    (* Table initialization: fTable_Al *)
    fTable_Al[0, 0] := 10.0000; fTable_Al[0, 1] := -9999; fTable_Al[0, 2] := 3.11990;
    fTable_Al[1, 0] := 10.1617; fTable_Al[1, 1] := -9999; fTable_Al[1, 2] := 3.05822;
    fTable_Al[2, 0] := 10.3261; fTable_Al[2, 1] := -9999; fTable_Al[2, 2] := 2.99776;
    fTable_Al[3, 0] := 10.4931; fTable_Al[3, 1] := -9999; fTable_Al[3, 2] := 2.93850;
    fTable_Al[4, 0] := 10.6628; fTable_Al[4, 1] := -9999; fTable_Al[4, 2] := 2.88041;
    fTable_Al[5, 0] := 10.8353; fTable_Al[5, 1] := -9999; fTable_Al[5, 2] := 2.82347;
    fTable_Al[6, 0] := 11.0106; fTable_Al[6, 1] := -9999; fTable_Al[6, 2] := 2.76766;
    fTable_Al[7, 0] := 11.1886; fTable_Al[7, 1] := -9999; fTable_Al[7, 2] := 2.72200;
    fTable_Al[8, 0] := 11.3696; fTable_Al[8, 1] := -9999; fTable_Al[8, 2] := 2.69148;
    fTable_Al[9, 0] := 11.5535; fTable_Al[9, 1] := -9999; fTable_Al[9, 2] := 2.66129;
    fTable_Al[10, 0] := 11.7404; fTable_Al[10, 1] := -9999; fTable_Al[10, 2] := 2.63145;
    fTable_Al[11, 0] := 11.9303; fTable_Al[11, 1] := -9999; fTable_Al[11, 2] := 2.60195;
    fTable_Al[12, 0] := 12.1232; fTable_Al[12, 1] := -9999; fTable_Al[12, 2] := 2.57277;
    fTable_Al[13, 0] := 12.3193; fTable_Al[13, 1] := -9999; fTable_Al[13, 2] := 2.54392;
    fTable_Al[14, 0] := 12.5186; fTable_Al[14, 1] := -9999; fTable_Al[14, 2] := 2.51539;
    fTable_Al[15, 0] := 12.7210; fTable_Al[15, 1] := -9999; fTable_Al[15, 2] := 2.46668;
    fTable_Al[16, 0] := 12.9268; fTable_Al[16, 1] := -9999; fTable_Al[16, 2] := 2.41373;
    fTable_Al[17, 0] := 13.1359; fTable_Al[17, 1] := -9999; fTable_Al[17, 2] := 2.36192;
    fTable_Al[18, 0] := 13.3483; fTable_Al[18, 1] := -9999; fTable_Al[18, 2] := 2.30898;
    fTable_Al[19, 0] := 13.5642; fTable_Al[19, 1] := -9999; fTable_Al[19, 2] := 2.23405;
    fTable_Al[20, 0] := 13.7836; fTable_Al[20, 1] := -9999; fTable_Al[20, 2] := 2.15356;
    fTable_Al[21, 0] := 14.0066; fTable_Al[21, 1] := -9999; fTable_Al[21, 2] := 2.06069;
    fTable_Al[22, 0] := 14.2331; fTable_Al[22, 1] := -9999; fTable_Al[22, 2] := 1.96756;
    fTable_Al[23, 0] := 14.4633; fTable_Al[23, 1] := -9999; fTable_Al[23, 2] := 1.81305;
    fTable_Al[24, 0] := 14.6973; fTable_Al[24, 1] := -9999; fTable_Al[24, 2] := 1.35947;
    fTable_Al[25, 0] := 14.9350; fTable_Al[25, 1] := -9999; fTable_Al[25, 2] := 0.902011;
    fTable_Al[26, 0] := 15.1765; fTable_Al[26, 1] := -9999; fTable_Al[26, 2] := 0.609172;
    fTable_Al[27, 0] := 15.4220; fTable_Al[27, 1] := -9999; fTable_Al[27, 2] := 0.439681;
    fTable_Al[28, 0] := 15.6714; fTable_Al[28, 1] := -9999; fTable_Al[28, 2] := 0.372037;
    fTable_Al[29, 0] := 15.9249; fTable_Al[29, 1] := -9999; fTable_Al[29, 2] := 0.326005;
    fTable_Al[30, 0] := 16.1825; fTable_Al[30, 1] := -9999; fTable_Al[30, 2] := 0.285669;
    fTable_Al[31, 0] := 16.4442; fTable_Al[31, 1] := -9999; fTable_Al[31, 2] := 0.247205;
    fTable_Al[32, 0] := 16.7102; fTable_Al[32, 1] := -9999; fTable_Al[32, 2] := 0.213520;
    fTable_Al[33, 0] := 16.9805; fTable_Al[33, 1] := -9999; fTable_Al[33, 2] := 0.196522;
    fTable_Al[34, 0] := 17.2551; fTable_Al[34, 1] := -9999; fTable_Al[34, 2] := 0.181095;
    fTable_Al[35, 0] := 17.5342; fTable_Al[35, 1] := -9999; fTable_Al[35, 2] := 0.168385;
    fTable_Al[36, 0] := 17.8178; fTable_Al[36, 1] := -9999; fTable_Al[36, 2] := 0.160808;
    fTable_Al[37, 0] := 18.1060; fTable_Al[37, 1] := -9999; fTable_Al[37, 2] := 0.153573;
    fTable_Al[38, 0] := 18.3989; fTable_Al[38, 1] := -9999; fTable_Al[38, 2] := 0.146663;
    fTable_Al[39, 0] := 18.6964; fTable_Al[39, 1] := -9999; fTable_Al[39, 2] := 0.140063;
    fTable_Al[40, 0] := 18.9988; fTable_Al[40, 1] := -9999; fTable_Al[40, 2] := 0.133164;
    fTable_Al[41, 0] := 19.3061; fTable_Al[41, 1] := -9999; fTable_Al[41, 2] := 0.126575;
    fTable_Al[42, 0] := 19.6184; fTable_Al[42, 1] := -9999; fTable_Al[42, 2] := 0.120312;
    fTable_Al[43, 0] := 19.9357; fTable_Al[43, 1] := -9999; fTable_Al[43, 2] := 0.114360;
    fTable_Al[44, 0] := 20.2582; fTable_Al[44, 1] := -9999; fTable_Al[44, 2] := 0.109752;
    fTable_Al[45, 0] := 20.5858; fTable_Al[45, 1] := -9999; fTable_Al[45, 2] := 0.111010;
    fTable_Al[46, 0] := 20.9188; fTable_Al[46, 1] := -9999; fTable_Al[46, 2] := 0.112282;
    fTable_Al[47, 0] := 21.2571; fTable_Al[47, 1] := -9999; fTable_Al[47, 2] := 0.113569;
    fTable_Al[48, 0] := 21.6009; fTable_Al[48, 1] := -9999; fTable_Al[48, 2] := 0.114870;
    fTable_Al[49, 0] := 21.9503; fTable_Al[49, 1] := -9999; fTable_Al[49, 2] := 0.116186;
    fTable_Al[50, 0] := 22.3053; fTable_Al[50, 1] := -9999; fTable_Al[50, 2] := 0.117518;
    fTable_Al[51, 0] := 22.6661; fTable_Al[51, 1] := -9999; fTable_Al[51, 2] := 0.118864;
    fTable_Al[52, 0] := 23.0327; fTable_Al[52, 1] := -9999; fTable_Al[52, 2] := 0.120227;
    fTable_Al[53, 0] := 23.4053; fTable_Al[53, 1] := -9999; fTable_Al[53, 2] := 0.122751;
    fTable_Al[54, 0] := 23.7838; fTable_Al[54, 1] := -9999; fTable_Al[54, 2] := 0.126315;
    fTable_Al[55, 0] := 24.1685; fTable_Al[55, 1] := -9999; fTable_Al[55, 2] := 0.129984;
    fTable_Al[56, 0] := 24.5594; fTable_Al[56, 1] := -9999; fTable_Al[56, 2] := 0.133759;
    fTable_Al[57, 0] := 24.9566; fTable_Al[57, 1] := -9999; fTable_Al[57, 2] := 0.137643;
    fTable_Al[58, 0] := 25.3603; fTable_Al[58, 1] := -9999; fTable_Al[58, 2] := 0.141640;
    fTable_Al[59, 0] := 25.7705; fTable_Al[59, 1] := -9999; fTable_Al[59, 2] := 0.145495;
    fTable_Al[60, 0] := 26.1873; fTable_Al[60, 1] := -9999; fTable_Al[60, 2] := 0.148244;
    fTable_Al[61, 0] := 26.6109; fTable_Al[61, 1] := -9999; fTable_Al[61, 2] := 0.151045;
    fTable_Al[62, 0] := 27.0413; fTable_Al[62, 1] := -9999; fTable_Al[62, 2] := 0.153898;
    fTable_Al[63, 0] := 27.4786; fTable_Al[63, 1] := -9999; fTable_Al[63, 2] := 0.156806;
    fTable_Al[64, 0] := 27.9231; fTable_Al[64, 1] := -9999; fTable_Al[64, 2] := 0.159768;
    fTable_Al[65, 0] := 28.3747; fTable_Al[65, 1] := -9999; fTable_Al[65, 2] := 0.162787;
    fTable_Al[66, 0] := 28.8337; fTable_Al[66, 1] := -9999; fTable_Al[66, 2] := 0.165863;
    fTable_Al[67, 0] := 29.3000; fTable_Al[67, 1] := 2.34285; fTable_Al[67, 2] := 0.168996;
    fTable_Al[68, 0] := 29.7739; fTable_Al[68, 1] := 2.32717; fTable_Al[68, 2] := 0.172189;
    fTable_Al[69, 0] := 30.2555; fTable_Al[69, 1] := 2.31139; fTable_Al[69, 2] := 0.175442;
    fTable_Al[70, 0] := 30.7449; fTable_Al[70, 1] := 2.29552; fTable_Al[70, 2] := 0.178757;
    fTable_Al[71, 0] := 31.2421; fTable_Al[71, 1] := 2.27956; fTable_Al[71, 2] := 0.182134;
    fTable_Al[72, 0] := 31.7475; fTable_Al[72, 1] := 2.26350; fTable_Al[72, 2] := 0.185575;
    fTable_Al[73, 0] := 32.2609; fTable_Al[73, 1] := 2.24754; fTable_Al[73, 2] := 0.189081;
    fTable_Al[74, 0] := 32.7827; fTable_Al[74, 1] := 2.23175; fTable_Al[74, 2] := 0.192378;
    fTable_Al[75, 0] := 33.3130; fTable_Al[75, 1] := 2.21555; fTable_Al[75, 2] := 0.194561;
    fTable_Al[76, 0] := 33.8518; fTable_Al[76, 1] := 2.19843; fTable_Al[76, 2] := 0.196767;
    fTable_Al[77, 0] := 34.3993; fTable_Al[77, 1] := 2.18068; fTable_Al[77, 2] := 0.198999;
    fTable_Al[78, 0] := 34.9557; fTable_Al[78, 1] := 2.16235; fTable_Al[78, 2] := 0.201256;
    fTable_Al[79, 0] := 35.5211; fTable_Al[79, 1] := 2.14342; fTable_Al[79, 2] := 0.203539;
    fTable_Al[80, 0] := 36.0956; fTable_Al[80, 1] := 2.12388; fTable_Al[80, 2] := 0.205847;
    fTable_Al[81, 0] := 36.6794; fTable_Al[81, 1] := 2.10371; fTable_Al[81, 2] := 0.208182;
    fTable_Al[82, 0] := 37.2727; fTable_Al[82, 1] := 2.08287; fTable_Al[82, 2] := 0.210544;
    fTable_Al[83, 0] := 37.8755; fTable_Al[83, 1] := 2.06135; fTable_Al[83, 2] := 0.212932;
    fTable_Al[84, 0] := 38.4882; fTable_Al[84, 1] := 2.03911; fTable_Al[84, 2] := 0.215347;
    fTable_Al[85, 0] := 39.1107; fTable_Al[85, 1] := 2.01612; fTable_Al[85, 2] := 0.217789;
    fTable_Al[86, 0] := 39.7432; fTable_Al[86, 1] := 1.99237; fTable_Al[86, 2] := 0.220259;
    fTable_Al[87, 0] := 40.3861; fTable_Al[87, 1] := 1.96797; fTable_Al[87, 2] := 0.222758;
    fTable_Al[88, 0] := 41.0393; fTable_Al[88, 1] := 1.94295; fTable_Al[88, 2] := 0.225068;
    fTable_Al[89, 0] := 41.7031; fTable_Al[89, 1] := 1.91682; fTable_Al[89, 2] := 0.226470;
    fTable_Al[90, 0] := 42.3776; fTable_Al[90, 1] := 1.88912; fTable_Al[90, 2] := 0.227880;
    fTable_Al[91, 0] := 43.0630; fTable_Al[91, 1] := 1.86007; fTable_Al[91, 2] := 0.229299;
    fTable_Al[92, 0] := 43.7595; fTable_Al[92, 1] := 1.82966; fTable_Al[92, 2] := 0.230727;
    fTable_Al[93, 0] := 44.4673; fTable_Al[93, 1] := 1.79787; fTable_Al[93, 2] := 0.232164;
    fTable_Al[94, 0] := 45.1865; fTable_Al[94, 1] := 1.76466; fTable_Al[94, 2] := 0.233610;
    fTable_Al[95, 0] := 45.9174; fTable_Al[95, 1] := 1.73005; fTable_Al[95, 2] := 0.235064;
    fTable_Al[96, 0] := 46.6600; fTable_Al[96, 1] := 1.69399; fTable_Al[96, 2] := 0.236528;
    fTable_Al[97, 0] := 47.4147; fTable_Al[97, 1] := 1.65814; fTable_Al[97, 2] := 0.238001;
    fTable_Al[98, 0] := 48.1816; fTable_Al[98, 1] := 1.62074; fTable_Al[98, 2] := 0.235842;
    fTable_Al[99, 0] := 48.9609; fTable_Al[99, 1] := 1.57843; fTable_Al[99, 2] := 0.232104;
    fTable_Al[100, 0] := 49.7528; fTable_Al[100, 1] := 1.53229; fTable_Al[100, 2] := 0.228425;
    fTable_Al[101, 0] := 50.5576; fTable_Al[101, 1] := 1.48252; fTable_Al[101, 2] := 0.224805;
    fTable_Al[102, 0] := 51.3753; fTable_Al[102, 1] := 1.42904; fTable_Al[102, 2] := 0.221242;
    fTable_Al[103, 0] := 52.2062; fTable_Al[103, 1] := 1.37159; fTable_Al[103, 2] := 0.217735;
    fTable_Al[104, 0] := 53.0506; fTable_Al[104, 1] := 1.30972; fTable_Al[104, 2] := 0.214284;
    fTable_Al[105, 0] := 53.9087; fTable_Al[105, 1] := 1.24315; fTable_Al[105, 2] := 0.211759;
    fTable_Al[106, 0] := 54.7806; fTable_Al[106, 1] := 1.17229; fTable_Al[106, 2] := 0.209829;
    fTable_Al[107, 0] := 55.6667; fTable_Al[107, 1] := 1.09675; fTable_Al[107, 2] := 0.207917;
    fTable_Al[108, 0] := 56.5670; fTable_Al[108, 1] := 1.01559; fTable_Al[108, 2] := 0.206022;
    fTable_Al[109, 0] := 57.4820; fTable_Al[109, 1] := 0.928103; fTable_Al[109, 2] := 0.204145;
    fTable_Al[110, 0] := 58.4117; fTable_Al[110, 1] := 0.833427; fTable_Al[110, 2] := 0.202284;
    fTable_Al[111, 0] := 59.3564; fTable_Al[111, 1] := 0.729805; fTable_Al[111, 2] := 0.200441;
    fTable_Al[112, 0] := 60.3165; fTable_Al[112, 1] := 0.616720; fTable_Al[112, 2] := 0.200207;
    fTable_Al[113, 0] := 61.2921; fTable_Al[113, 1] := 0.494009; fTable_Al[113, 2] := 0.200602;
    fTable_Al[114, 0] := 62.2834; fTable_Al[114, 1] := 0.359171; fTable_Al[114, 2] := 0.200998;
    fTable_Al[115, 0] := 63.2908; fTable_Al[115, 1] := 0.206766; fTable_Al[115, 2] := 0.201394;
    fTable_Al[116, 0] := 64.3145; fTable_Al[116, 1] := 0.0367838; fTable_Al[116, 2] := 0.208215;
    fTable_Al[117, 0] := 65.3547; fTable_Al[117, 1] := -0.150100; fTable_Al[117, 2] := 0.215821;
    fTable_Al[118, 0] := 66.4118; fTable_Al[118, 1] := -0.363400; fTable_Al[118, 2] := 0.223705;
    fTable_Al[119, 0] := 67.4859; fTable_Al[119, 1] := -0.612251; fTable_Al[119, 2] := 0.231878;
    fTable_Al[120, 0] := 68.5775; fTable_Al[120, 1] := -0.913185; fTable_Al[120, 2] := 0.239512;
    fTable_Al[121, 0] := 69.6867; fTable_Al[121, 1] := -1.29772; fTable_Al[121, 2] := 0.247287;
    fTable_Al[122, 0] := 70.8138; fTable_Al[122, 1] := -1.83916; fTable_Al[122, 2] := 0.255315;
    fTable_Al[123, 0] := 71.9591; fTable_Al[123, 1] := -2.82640; fTable_Al[123, 2] := 0.263603;
    fTable_Al[124, 0] := 72.6000; fTable_Al[124, 1] := -4.71870; fTable_Al[124, 2] := 0.268298;
    fTable_Al[125, 0] := 72.8000; fTable_Al[125, 1] := -4.77865; fTable_Al[125, 2] := 3.05391;
    fTable_Al[126, 0] := 73.1230; fTable_Al[126, 1] := -3.57738; fTable_Al[126, 2] := 3.10106;
    fTable_Al[127, 0] := 74.3057; fTable_Al[127, 1] := -2.58986; fTable_Al[127, 2] := 3.27808;
    fTable_Al[128, 0] := 75.5076; fTable_Al[128, 1] := -2.24498; fTable_Al[128, 2] := 3.46521;
    fTable_Al[129, 0] := 76.7289; fTable_Al[129, 1] := -2.04974; fTable_Al[129, 2] := 3.66301;
    fTable_Al[130, 0] := 77.9699; fTable_Al[130, 1] := -1.91658; fTable_Al[130, 2] := 3.87212;
    fTable_Al[131, 0] := 79.2310; fTable_Al[131, 1] := -1.81173; fTable_Al[131, 2] := 4.09316;
    fTable_Al[132, 0] := 80.5125; fTable_Al[132, 1] := -1.71207; fTable_Al[132, 2] := 4.32681;
    fTable_Al[133, 0] := 81.8147; fTable_Al[133, 1] := -1.61278; fTable_Al[133, 2] := 4.55877;
    fTable_Al[134, 0] := 83.1380; fTable_Al[134, 1] := -1.51695; fTable_Al[134, 2] := 4.80227;
    fTable_Al[135, 0] := 84.4827; fTable_Al[135, 1] := -1.40821; fTable_Al[135, 2] := 5.05877;
    fTable_Al[136, 0] := 85.8491; fTable_Al[136, 1] := -1.24639; fTable_Al[136, 2] := 5.32897;
    fTable_Al[137, 0] := 87.2377; fTable_Al[137, 1] := -1.04412; fTable_Al[137, 2] := 5.54566;
    fTable_Al[138, 0] := 88.6487; fTable_Al[138, 1] := -0.869623; fTable_Al[138, 2] := 5.69070;
    fTable_Al[139, 0] := 90.0825; fTable_Al[139, 1] := -0.729715; fTable_Al[139, 2] := 5.83953;
    fTable_Al[140, 0] := 91.5395; fTable_Al[140, 1] := -0.602517; fTable_Al[140, 2] := 5.99225;
    fTable_Al[141, 0] := 93.0201; fTable_Al[141, 1] := -0.481649; fTable_Al[141, 2] := 6.14897;
    fTable_Al[142, 0] := 94.5246; fTable_Al[142, 1] := -0.363849; fTable_Al[142, 2] := 6.30978;
    fTable_Al[143, 0] := 96.0535; fTable_Al[143, 1] := -0.246485; fTable_Al[143, 2] := 6.47480;
    fTable_Al[144, 0] := 97.6071; fTable_Al[144, 1] := -0.127798; fTable_Al[144, 2] := 6.64413;
    fTable_Al[145, 0] := 99.1858; fTable_Al[145, 1] := -0.00572152; fTable_Al[145, 2] := 6.81790;
    fTable_Al[146, 0] := 100.790; fTable_Al[146, 1] := 0.121587; fTable_Al[146, 2] := 6.99620;
    fTable_Al[147, 0] := 102.420; fTable_Al[147, 1] := 0.257648; fTable_Al[147, 2] := 7.17918;
    fTable_Al[148, 0] := 104.077; fTable_Al[148, 1] := 0.408417; fTable_Al[148, 2] := 7.36022;
    fTable_Al[149, 0] := 105.760; fTable_Al[149, 1] := 0.563135; fTable_Al[149, 2] := 7.52866;
    fTable_Al[150, 0] := 107.471; fTable_Al[150, 1] := 0.713525; fTable_Al[150, 2] := 7.70096;
    fTable_Al[151, 0] := 109.209; fTable_Al[151, 1] := 0.869599; fTable_Al[151, 2] := 7.87720;
    fTable_Al[152, 0] := 110.975; fTable_Al[152, 1] := 1.03257; fTable_Al[152, 2] := 8.05748;
    fTable_Al[153, 0] := 112.770; fTable_Al[153, 1] := 1.20465; fTable_Al[153, 2] := 8.24188;
    fTable_Al[154, 0] := 114.594; fTable_Al[154, 1] := 1.38785; fTable_Al[154, 2] := 8.43050;
    fTable_Al[155, 0] := 116.448; fTable_Al[155, 1] := 1.58511; fTable_Al[155, 2] := 8.62344;
    fTable_Al[156, 0] := 118.331; fTable_Al[156, 1] := 1.79993; fTable_Al[156, 2] := 8.82080;
    fTable_Al[157, 0] := 120.245; fTable_Al[157, 1] := 2.03832; fTable_Al[157, 2] := 9.02267;
    fTable_Al[158, 0] := 122.190; fTable_Al[158, 1] := 2.31105; fTable_Al[158, 2] := 9.22916;
    fTable_Al[159, 0] := 124.166; fTable_Al[159, 1] := 2.65726; fTable_Al[159, 2] := 9.44037;
    fTable_Al[160, 0] := 126.175; fTable_Al[160, 1] := 3.05450; fTable_Al[160, 2] := 9.49754;
    fTable_Al[161, 0] := 128.215; fTable_Al[161, 1] := 3.37636; fTable_Al[161, 2] := 9.51114;
    fTable_Al[162, 0] := 130.289; fTable_Al[162, 1] := 3.65455; fTable_Al[162, 2] := 9.52475;
    fTable_Al[163, 0] := 132.397; fTable_Al[163, 1] := 3.91635; fTable_Al[163, 2] := 9.53840;
    fTable_Al[164, 0] := 134.538; fTable_Al[164, 1] := 4.16654; fTable_Al[164, 2] := 9.55206;
    fTable_Al[165, 0] := 136.714; fTable_Al[165, 1] := 4.40886; fTable_Al[165, 2] := 9.56573;
    fTable_Al[166, 0] := 138.925; fTable_Al[166, 1] := 4.64594; fTable_Al[166, 2] := 9.57943;
    fTable_Al[167, 0] := 141.172; fTable_Al[167, 1] := 4.87987; fTable_Al[167, 2] := 9.59315;
    fTable_Al[168, 0] := 143.456; fTable_Al[168, 1] := 5.11258; fTable_Al[168, 2] := 9.60689;
    fTable_Al[169, 0] := 145.776; fTable_Al[169, 1] := 5.34618; fTable_Al[169, 2] := 9.62064;
    fTable_Al[170, 0] := 148.134; fTable_Al[170, 1] := 5.58438; fTable_Al[170, 2] := 9.63443;
    fTable_Al[171, 0] := 150.530; fTable_Al[171, 1] := 5.83549; fTable_Al[171, 2] := 9.64822;
    fTable_Al[172, 0] := 152.964; fTable_Al[172, 1] := 6.09089; fTable_Al[172, 2] := 9.62310;
    fTable_Al[173, 0] := 155.439; fTable_Al[173, 1] := 6.32655; fTable_Al[173, 2] := 9.59689;
    fTable_Al[174, 0] := 157.953; fTable_Al[174, 1] := 6.55613; fTable_Al[174, 2] := 9.57075;
    fTable_Al[175, 0] := 160.507; fTable_Al[175, 1] := 6.78302; fTable_Al[175, 2] := 9.54468;
    fTable_Al[176, 0] := 163.103; fTable_Al[176, 1] := 7.00948; fTable_Al[176, 2] := 9.51868;
    fTable_Al[177, 0] := 165.742; fTable_Al[177, 1] := 7.23759; fTable_Al[177, 2] := 9.49275;
    fTable_Al[178, 0] := 168.422; fTable_Al[178, 1] := 7.46980; fTable_Al[178, 2] := 9.46689;
    fTable_Al[179, 0] := 171.146; fTable_Al[179, 1] := 7.70942; fTable_Al[179, 2] := 9.44111;
    fTable_Al[180, 0] := 173.915; fTable_Al[180, 1] := 7.96219; fTable_Al[180, 2] := 9.41540;
    fTable_Al[181, 0] := 176.727; fTable_Al[181, 1] := 8.24313; fTable_Al[181, 2] := 9.38975;
    fTable_Al[182, 0] := 179.586; fTable_Al[182, 1] := 8.57964; fTable_Al[182, 2] := 9.31472;
    fTable_Al[183, 0] := 182.491; fTable_Al[183, 1] := 8.88946; fTable_Al[183, 2] := 9.13115;
    fTable_Al[184, 0] := 185.442; fTable_Al[184, 1] := 9.11623; fTable_Al[184, 2] := 8.95119;
    fTable_Al[185, 0] := 188.442; fTable_Al[185, 1] := 9.32069; fTable_Al[185, 2] := 8.77477;
    fTable_Al[186, 0] := 191.489; fTable_Al[186, 1] := 9.50496; fTable_Al[186, 2] := 8.60184;
    fTable_Al[187, 0] := 194.587; fTable_Al[187, 1] := 9.67311; fTable_Al[187, 2] := 8.43231;
    fTable_Al[188, 0] := 197.734; fTable_Al[188, 1] := 9.82798; fTable_Al[188, 2] := 8.26612;
    fTable_Al[189, 0] := 200.932; fTable_Al[189, 1] := 9.97197; fTable_Al[189, 2] := 8.10317;
    fTable_Al[190, 0] := 204.182; fTable_Al[190, 1] := 10.1053; fTable_Al[190, 2] := 7.93953;
    fTable_Al[191, 0] := 207.485; fTable_Al[191, 1] := 10.2265; fTable_Al[191, 2] := 7.77920;
    fTable_Al[192, 0] := 210.840; fTable_Al[192, 1] := 10.3376; fTable_Al[192, 2] := 7.62210;
    fTable_Al[193, 0] := 214.251; fTable_Al[193, 1] := 10.4388; fTable_Al[193, 2] := 7.46817;
    fTable_Al[194, 0] := 217.716; fTable_Al[194, 1] := 10.5299; fTable_Al[194, 2] := 7.31736;
    fTable_Al[195, 0] := 221.237; fTable_Al[195, 1] := 10.6083; fTable_Al[195, 2] := 7.16959;
    fTable_Al[196, 0] := 224.816; fTable_Al[196, 1] := 10.6680; fTable_Al[196, 2] := 7.03532;
    fTable_Al[197, 0] := 228.452; fTable_Al[197, 1] := 10.7284; fTable_Al[197, 2] := 6.92993;
    fTable_Al[198, 0] := 232.147; fTable_Al[198, 1] := 10.8042; fTable_Al[198, 2] := 6.82611;
    fTable_Al[199, 0] := 235.902; fTable_Al[199, 1] := 10.8811; fTable_Al[199, 2] := 6.72384;
    fTable_Al[200, 0] := 239.717; fTable_Al[200, 1] := 10.9592; fTable_Al[200, 2] := 6.62312;
    fTable_Al[201, 0] := 243.595; fTable_Al[201, 1] := 11.0380; fTable_Al[201, 2] := 6.52389;
    fTable_Al[202, 0] := 247.535; fTable_Al[202, 1] := 11.1176; fTable_Al[202, 2] := 6.42616;
    fTable_Al[203, 0] := 251.538; fTable_Al[203, 1] := 11.1983; fTable_Al[203, 2] := 6.32988;
    fTable_Al[204, 0] := 255.607; fTable_Al[204, 1] := 11.2808; fTable_Al[204, 2] := 6.23505;
    fTable_Al[205, 0] := 259.741; fTable_Al[205, 1] := 11.3664; fTable_Al[205, 2] := 6.14164;
    fTable_Al[206, 0] := 263.942; fTable_Al[206, 1] := 11.4630; fTable_Al[206, 2] := 6.04964;
    fTable_Al[207, 0] := 268.211; fTable_Al[207, 1] := 11.5725; fTable_Al[207, 2] := 5.94856;
    fTable_Al[208, 0] := 272.549; fTable_Al[208, 1] := 11.6747; fTable_Al[208, 2] := 5.80523;
    fTable_Al[209, 0] := 276.957; fTable_Al[209, 1] := 11.7511; fTable_Al[209, 2] := 5.66535;
    fTable_Al[210, 0] := 281.437; fTable_Al[210, 1] := 11.8159; fTable_Al[210, 2] := 5.52884;
    fTable_Al[211, 0] := 285.989; fTable_Al[211, 1] := 11.8724; fTable_Al[211, 2] := 5.39563;
    fTable_Al[212, 0] := 290.615; fTable_Al[212, 1] := 11.9222; fTable_Al[212, 2] := 5.26561;
    fTable_Al[213, 0] := 295.315; fTable_Al[213, 1] := 11.9664; fTable_Al[213, 2] := 5.13874;
    fTable_Al[214, 0] := 300.092; fTable_Al[214, 1] := 12.0058; fTable_Al[214, 2] := 5.01492;
    fTable_Al[215, 0] := 304.945; fTable_Al[215, 1] := 12.0408; fTable_Al[215, 2] := 4.89409;
    fTable_Al[216, 0] := 309.878; fTable_Al[216, 1] := 12.0718; fTable_Al[216, 2] := 4.77616;
    fTable_Al[217, 0] := 314.890; fTable_Al[217, 1] := 12.0993; fTable_Al[217, 2] := 4.66108;
    fTable_Al[218, 0] := 319.983; fTable_Al[218, 1] := 12.1235; fTable_Al[218, 2] := 4.54877;
    fTable_Al[219, 0] := 325.158; fTable_Al[219, 1] := 12.1445; fTable_Al[219, 2] := 4.43917;
    fTable_Al[220, 0] := 330.418; fTable_Al[220, 1] := 12.1625; fTable_Al[220, 2] := 4.33221;
    fTable_Al[221, 0] := 335.762; fTable_Al[221, 1] := 12.1777; fTable_Al[221, 2] := 4.22782;
    fTable_Al[222, 0] := 341.192; fTable_Al[222, 1] := 12.1900; fTable_Al[222, 2] := 4.12595;
    fTable_Al[223, 0] := 346.711; fTable_Al[223, 1] := 12.1992; fTable_Al[223, 2] := 4.02654;
    fTable_Al[224, 0] := 352.319; fTable_Al[224, 1] := 12.2049; fTable_Al[224, 2] := 3.92952;
    fTable_Al[225, 0] := 358.017; fTable_Al[225, 1] := 12.2045; fTable_Al[225, 2] := 3.83484;
    fTable_Al[226, 0] := 363.808; fTable_Al[226, 1] := 12.1998; fTable_Al[226, 2] := 3.75388;
    fTable_Al[227, 0] := 369.692; fTable_Al[227, 1] := 12.2008; fTable_Al[227, 2] := 3.67818;
    fTable_Al[228, 0] := 375.672; fTable_Al[228, 1] := 12.2048; fTable_Al[228, 2] := 3.60400;
    fTable_Al[229, 0] := 381.748; fTable_Al[229, 1] := 12.2097; fTable_Al[229, 2] := 3.53133;
    fTable_Al[230, 0] := 387.922; fTable_Al[230, 1] := 12.2152; fTable_Al[230, 2] := 3.46011;
    fTable_Al[231, 0] := 394.197; fTable_Al[231, 1] := 12.2210; fTable_Al[231, 2] := 3.39034;
    fTable_Al[232, 0] := 400.573; fTable_Al[232, 1] := 12.2270; fTable_Al[232, 2] := 3.32197;
    fTable_Al[233, 0] := 407.052; fTable_Al[233, 1] := 12.2333; fTable_Al[233, 2] := 3.25498;
    fTable_Al[234, 0] := 413.635; fTable_Al[234, 1] := 12.2399; fTable_Al[234, 2] := 3.18934;
    fTable_Al[235, 0] := 420.326; fTable_Al[235, 1] := 12.2470; fTable_Al[235, 2] := 3.12502;
    fTable_Al[236, 0] := 427.124; fTable_Al[236, 1] := 12.2549; fTable_Al[236, 2] := 3.06201;
    fTable_Al[237, 0] := 434.032; fTable_Al[237, 1] := 12.2652; fTable_Al[237, 2] := 3.00026;
    fTable_Al[238, 0] := 441.052; fTable_Al[238, 1] := 12.2773; fTable_Al[238, 2] := 2.93296;
    fTable_Al[239, 0] := 448.186; fTable_Al[239, 1] := 12.2849; fTable_Al[239, 2] := 2.86424;
    fTable_Al[240, 0] := 455.435; fTable_Al[240, 1] := 12.2892; fTable_Al[240, 2] := 2.79730;
    fTable_Al[241, 0] := 462.802; fTable_Al[241, 1] := 12.2920; fTable_Al[241, 2] := 2.73189;
    fTable_Al[242, 0] := 470.287; fTable_Al[242, 1] := 12.2937; fTable_Al[242, 2] := 2.66798;
    fTable_Al[243, 0] := 477.894; fTable_Al[243, 1] := 12.2943; fTable_Al[243, 2] := 2.60559;
    fTable_Al[244, 0] := 485.623; fTable_Al[244, 1] := 12.2945; fTable_Al[244, 2] := 2.54463;
    fTable_Al[245, 0] := 493.478; fTable_Al[245, 1] := 12.2942; fTable_Al[245, 2] := 2.48490;
    fTable_Al[246, 0] := 501.459; fTable_Al[246, 1] := 12.2939; fTable_Al[246, 2] := 2.42570;
    fTable_Al[247, 0] := 509.570; fTable_Al[247, 1] := 12.2928; fTable_Al[247, 2] := 2.36643;
    fTable_Al[248, 0] := 517.812; fTable_Al[248, 1] := 12.2896; fTable_Al[248, 2] := 2.30801;
    fTable_Al[249, 0] := 526.187; fTable_Al[249, 1] := 12.2852; fTable_Al[249, 2] := 2.25125;
    fTable_Al[250, 0] := 534.698; fTable_Al[250, 1] := 12.2801; fTable_Al[250, 2] := 2.19625;
    fTable_Al[251, 0] := 543.346; fTable_Al[251, 1] := 12.2748; fTable_Al[251, 2] := 2.14277;
    fTable_Al[252, 0] := 552.134; fTable_Al[252, 1] := 12.2700; fTable_Al[252, 2] := 2.09062;
    fTable_Al[253, 0] := 561.065; fTable_Al[253, 1] := 12.2653; fTable_Al[253, 2] := 2.03805;
    fTable_Al[254, 0] := 570.139; fTable_Al[254, 1] := 12.2592; fTable_Al[254, 2] := 1.98589;
    fTable_Al[255, 0] := 579.361; fTable_Al[255, 1] := 12.2522; fTable_Al[255, 2] := 1.93406;
    fTable_Al[256, 0] := 588.732; fTable_Al[256, 1] := 12.2437; fTable_Al[256, 2] := 1.88338;
    fTable_Al[257, 0] := 598.254; fTable_Al[257, 1] := 12.2344; fTable_Al[257, 2] := 1.83389;
    fTable_Al[258, 0] := 607.930; fTable_Al[258, 1] := 12.2243; fTable_Al[258, 2] := 1.78571;
    fTable_Al[259, 0] := 617.763; fTable_Al[259, 1] := 12.2138; fTable_Al[259, 2] := 1.73879;
    fTable_Al[260, 0] := 627.755; fTable_Al[260, 1] := 12.2034; fTable_Al[260, 2] := 1.69298;
    fTable_Al[261, 0] := 637.908; fTable_Al[261, 1] := 12.1929; fTable_Al[261, 2] := 1.64704;
    fTable_Al[262, 0] := 648.226; fTable_Al[262, 1] := 12.1814; fTable_Al[262, 2] := 1.60038;
    fTable_Al[263, 0] := 658.711; fTable_Al[263, 1] := 12.1674; fTable_Al[263, 2] := 1.55377;
    fTable_Al[264, 0] := 669.365; fTable_Al[264, 1] := 12.1491; fTable_Al[264, 2] := 1.50856;
    fTable_Al[265, 0] := 680.191; fTable_Al[265, 1] := 12.1287; fTable_Al[265, 2] := 1.46882;
    fTable_Al[266, 0] := 691.193; fTable_Al[266, 1] := 12.1108; fTable_Al[266, 2] := 1.43328;
    fTable_Al[267, 0] := 702.372; fTable_Al[267, 1] := 12.0954; fTable_Al[267, 2] := 1.39941;
    fTable_Al[268, 0] := 713.733; fTable_Al[268, 1] := 12.0820; fTable_Al[268, 2] := 1.36380;
    fTable_Al[269, 0] := 725.277; fTable_Al[269, 1] := 12.0674; fTable_Al[269, 2] := 1.32737;
    fTable_Al[270, 0] := 737.008; fTable_Al[270, 1] := 12.0514; fTable_Al[270, 2] := 1.29193;
    fTable_Al[271, 0] := 748.928; fTable_Al[271, 1] := 12.0350; fTable_Al[271, 2] := 1.25742;
    fTable_Al[272, 0] := 761.042; fTable_Al[272, 1] := 12.0181; fTable_Al[272, 2] := 1.22382;
    fTable_Al[273, 0] := 773.351; fTable_Al[273, 1] := 12.0009; fTable_Al[273, 2] := 1.19100;
    fTable_Al[274, 0] := 785.859; fTable_Al[274, 1] := 11.9834; fTable_Al[274, 2] := 1.15872;
    fTable_Al[275, 0] := 798.570; fTable_Al[275, 1] := 11.9652; fTable_Al[275, 2] := 1.12705;
    fTable_Al[276, 0] := 811.486; fTable_Al[276, 1] := 11.9463; fTable_Al[276, 2] := 1.09624;
    fTable_Al[277, 0] := 824.611; fTable_Al[277, 1] := 11.9269; fTable_Al[277, 2] := 1.06625;
    fTable_Al[278, 0] := 837.949; fTable_Al[278, 1] := 11.9070; fTable_Al[278, 2] := 1.03708;
    fTable_Al[279, 0] := 851.502; fTable_Al[279, 1] := 11.8866; fTable_Al[279, 2] := 1.00870;
    fTable_Al[280, 0] := 865.274; fTable_Al[280, 1] := 11.8656; fTable_Al[280, 2] := 0.981035;
    fTable_Al[281, 0] := 879.269; fTable_Al[281, 1] := 11.8441; fTable_Al[281, 2] := 0.954065;
    fTable_Al[282, 0] := 893.491; fTable_Al[282, 1] := 11.8220; fTable_Al[282, 2] := 0.927842;
    fTable_Al[283, 0] := 907.943; fTable_Al[283, 1] := 11.7992; fTable_Al[283, 2] := 0.902346;
    fTable_Al[284, 0] := 922.628; fTable_Al[284, 1] := 11.7759; fTable_Al[284, 2] := 0.877557;
    fTable_Al[285, 0] := 937.551; fTable_Al[285, 1] := 11.7519; fTable_Al[285, 2] := 0.853321;
    fTable_Al[286, 0] := 952.715; fTable_Al[286, 1] := 11.7270; fTable_Al[286, 2] := 0.829761;
    fTable_Al[287, 0] := 968.124; fTable_Al[287, 1] := 11.7013; fTable_Al[287, 2] := 0.806859;
    fTable_Al[288, 0] := 983.783; fTable_Al[288, 1] := 11.6747; fTable_Al[288, 2] := 0.784555;
    fTable_Al[289, 0] := 999.695; fTable_Al[289, 1] := 11.6472; fTable_Al[289, 2] := 0.762967;
    fTable_Al[290, 0] := 1015.86; fTable_Al[290, 1] := 11.6184; fTable_Al[290, 2] := 0.742081;
    fTable_Al[291, 0] := 1032.29; fTable_Al[291, 1] := 11.5888; fTable_Al[291, 2] := 0.722661;
    fTable_Al[292, 0] := 1048.99; fTable_Al[292, 1] := 11.5591; fTable_Al[292, 2] := 0.703173;
    fTable_Al[293, 0] := 1065.96; fTable_Al[293, 1] := 11.5278; fTable_Al[293, 2] := 0.683588;
    fTable_Al[294, 0] := 1083.20; fTable_Al[294, 1] := 11.4947; fTable_Al[294, 2] := 0.664537;
    fTable_Al[295, 0] := 1100.72; fTable_Al[295, 1] := 11.4600; fTable_Al[295, 2] := 0.646018;
    fTable_Al[296, 0] := 1118.52; fTable_Al[296, 1] := 11.4234; fTable_Al[296, 2] := 0.628015;
    fTable_Al[297, 0] := 1136.61; fTable_Al[297, 1] := 11.3849; fTable_Al[297, 2] := 0.610519;
    fTable_Al[298, 0] := 1155; fTable_Al[298, 1] := 11.3440; fTable_Al[298, 2] := 0.593506;
    fTable_Al[299, 0] := 1173.68; fTable_Al[299, 1] := 11.3007; fTable_Al[299, 2] := 0.576965;
    fTable_Al[300, 0] := 1192.66; fTable_Al[300, 1] := 11.2544; fTable_Al[300, 2] := 0.560888;
    fTable_Al[301, 0] := 1211.95; fTable_Al[301, 1] := 11.2049; fTable_Al[301, 2] := 0.545258;
    fTable_Al[302, 0] := 1231.55; fTable_Al[302, 1] := 11.1516; fTable_Al[302, 2] := 0.530064;
    fTable_Al[303, 0] := 1251.47; fTable_Al[303, 1] := 11.0938; fTable_Al[303, 2] := 0.515441;
    fTable_Al[304, 0] := 1271.72; fTable_Al[304, 1] := 11.0310; fTable_Al[304, 2] := 0.501380;
    fTable_Al[305, 0] := 1292.29; fTable_Al[305, 1] := 10.9622; fTable_Al[305, 2] := 0.487892;
    fTable_Al[306, 0] := 1313.19; fTable_Al[306, 1] := 10.8865; fTable_Al[306, 2] := 0.474763;
    fTable_Al[307, 0] := 1334.43; fTable_Al[307, 1] := 10.8021; fTable_Al[307, 2] := 0.461987;
    fTable_Al[308, 0] := 1356.01; fTable_Al[308, 1] := 10.7069; fTable_Al[308, 2] := 0.449555;
    fTable_Al[309, 0] := 1377.94; fTable_Al[309, 1] := 10.5980; fTable_Al[309, 2] := 0.437459;
    fTable_Al[310, 0] := 1400.23; fTable_Al[310, 1] := 10.4713; fTable_Al[310, 2] := 0.425689;
    fTable_Al[311, 0] := 1422.88; fTable_Al[311, 1] := 10.3206; fTable_Al[311, 2] := 0.414239;
    fTable_Al[312, 0] := 1445.89; fTable_Al[312, 1] := 10.1361; fTable_Al[312, 2] := 0.403093;
    fTable_Al[313, 0] := 1469.28; fTable_Al[313, 1] := 9.90068; fTable_Al[313, 2] := 0.392100;
    fTable_Al[314, 0] := 1493.04; fTable_Al[314, 1] := 9.58044; fTable_Al[314, 2] := 0.381187;
    fTable_Al[315, 0] := 1517.19; fTable_Al[315, 1] := 9.09216; fTable_Al[315, 2] := 0.369680;
    fTable_Al[316, 0] := 1541.73; fTable_Al[316, 1] := 8.11537; fTable_Al[316, 2] := 0.358399;
    fTable_Al[317, 0] := 1559.50; fTable_Al[317, 1] := 1.89396; fTable_Al[317, 2] := 0.350553;
    fTable_Al[318, 0] := 1559.70; fTable_Al[318, 1] := 1.89589; fTable_Al[318, 2] := 4.16629;
    fTable_Al[319, 0] := 1566.67; fTable_Al[319, 1] := 7.10441; fTable_Al[319, 2] := 4.14105;
    fTable_Al[320, 0] := 1592.01; fTable_Al[320, 1] := 9.03572; fTable_Al[320, 2] := 4.05144;
    fTable_Al[321, 0] := 1617.76; fTable_Al[321, 1] := 9.80337; fTable_Al[321, 2] := 3.96379;
    fTable_Al[322, 0] := 1643.92; fTable_Al[322, 1] := 10.2995; fTable_Al[322, 2] := 3.87809;
    fTable_Al[323, 0] := 1670.51; fTable_Al[323, 1] := 10.6690; fTable_Al[323, 2] := 3.79420;
    fTable_Al[324, 0] := 1697.53; fTable_Al[324, 1] := 10.9642; fTable_Al[324, 2] := 3.71213;
    fTable_Al[325, 0] := 1724.99; fTable_Al[325, 1] := 11.2121; fTable_Al[325, 2] := 3.63182;
    fTable_Al[326, 0] := 1752.89; fTable_Al[326, 1] := 11.4254; fTable_Al[326, 2] := 3.54896;
    fTable_Al[327, 0] := 1781.24; fTable_Al[327, 1] := 11.6086; fTable_Al[327, 2] := 3.46653;
    fTable_Al[328, 0] := 1810.05; fTable_Al[328, 1] := 11.7695; fTable_Al[328, 2] := 3.38494;
    fTable_Al[329, 0] := 1839.32; fTable_Al[329, 1] := 11.9117; fTable_Al[329, 2] := 3.30527;
    fTable_Al[330, 0] := 1869.07; fTable_Al[330, 1] := 12.0391; fTable_Al[330, 2] := 3.22747;
    fTable_Al[331, 0] := 1899.30; fTable_Al[331, 1] := 12.1540; fTable_Al[331, 2] := 3.15148;
    fTable_Al[332, 0] := 1930.02; fTable_Al[332, 1] := 12.2583; fTable_Al[332, 2] := 3.07731;
    fTable_Al[333, 0] := 1961.24; fTable_Al[333, 1] := 12.3536; fTable_Al[333, 2] := 3.00489;
    fTable_Al[334, 0] := 1992.96; fTable_Al[334, 1] := 12.4408; fTable_Al[334, 2] := 2.93417;
    fTable_Al[335, 0] := 2025.20; fTable_Al[335, 1] := 12.5226; fTable_Al[335, 2] := 2.86696;
    fTable_Al[336, 0] := 2057.95; fTable_Al[336, 1] := 12.6001; fTable_Al[336, 2] := 2.79699;
    fTable_Al[337, 0] := 2091.24; fTable_Al[337, 1] := 12.6695; fTable_Al[337, 2] := 2.72803;
    fTable_Al[338, 0] := 2125.06; fTable_Al[338, 1] := 12.7334; fTable_Al[338, 2] := 2.66035;
    fTable_Al[339, 0] := 2159.43; fTable_Al[339, 1] := 12.7923; fTable_Al[339, 2] := 2.59405;
    fTable_Al[340, 0] := 2194.36; fTable_Al[340, 1] := 12.8467; fTable_Al[340, 2] := 2.52881;
    fTable_Al[341, 0] := 2229.85; fTable_Al[341, 1] := 12.8969; fTable_Al[341, 2] := 2.46498;
    fTable_Al[342, 0] := 2265.92; fTable_Al[342, 1] := 12.9433; fTable_Al[342, 2] := 2.40235;
    fTable_Al[343, 0] := 2302.57; fTable_Al[343, 1] := 12.9861; fTable_Al[343, 2] := 2.34101;
    fTable_Al[344, 0] := 2339.81; fTable_Al[344, 1] := 13.0257; fTable_Al[344, 2] := 2.28095;
    fTable_Al[345, 0] := 2377.66; fTable_Al[345, 1] := 13.0622; fTable_Al[345, 2] := 2.22204;
    fTable_Al[346, 0] := 2416.11; fTable_Al[346, 1] := 13.0960; fTable_Al[346, 2] := 2.16445;
    fTable_Al[347, 0] := 2455.19; fTable_Al[347, 1] := 13.1272; fTable_Al[347, 2] := 2.10810;
    fTable_Al[348, 0] := 2494.90; fTable_Al[348, 1] := 13.1560; fTable_Al[348, 2] := 2.05284;
    fTable_Al[349, 0] := 2535.26; fTable_Al[349, 1] := 13.1825; fTable_Al[349, 2] := 1.99885;
    fTable_Al[350, 0] := 2576.26; fTable_Al[350, 1] := 13.2068; fTable_Al[350, 2] := 1.94606;
    fTable_Al[351, 0] := 2617.93; fTable_Al[351, 1] := 13.2292; fTable_Al[351, 2] := 1.89447;
    fTable_Al[352, 0] := 2660.27; fTable_Al[352, 1] := 13.2498; fTable_Al[352, 2] := 1.84400;
    fTable_Al[353, 0] := 2703.30; fTable_Al[353, 1] := 13.2687; fTable_Al[353, 2] := 1.79474;
    fTable_Al[354, 0] := 2747.03; fTable_Al[354, 1] := 13.2859; fTable_Al[354, 2] := 1.74651;
    fTable_Al[355, 0] := 2791.46; fTable_Al[355, 1] := 13.3016; fTable_Al[355, 2] := 1.69945;
    fTable_Al[356, 0] := 2836.61; fTable_Al[356, 1] := 13.3159; fTable_Al[356, 2] := 1.65350;
    fTable_Al[357, 0] := 2882.49; fTable_Al[357, 1] := 13.3288; fTable_Al[357, 2] := 1.60862;
    fTable_Al[358, 0] := 2929.11; fTable_Al[358, 1] := 13.3405; fTable_Al[358, 2] := 1.56481;
    fTable_Al[359, 0] := 2976.48; fTable_Al[359, 1] := 13.3510; fTable_Al[359, 2] := 1.52204;
    fTable_Al[360, 0] := 3024.63; fTable_Al[360, 1] := 13.3604; fTable_Al[360, 2] := 1.48033;
    fTable_Al[361, 0] := 3073.55; fTable_Al[361, 1] := 13.3688; fTable_Al[361, 2] := 1.43961;
    fTable_Al[362, 0] := 3123.26; fTable_Al[362, 1] := 13.3762; fTable_Al[362, 2] := 1.39989;
    fTable_Al[363, 0] := 3173.78; fTable_Al[363, 1] := 13.3827; fTable_Al[363, 2] := 1.36116;
    fTable_Al[364, 0] := 3225.11; fTable_Al[364, 1] := 13.3883; fTable_Al[364, 2] := 1.32339;
    fTable_Al[365, 0] := 3277.27; fTable_Al[365, 1] := 13.3932; fTable_Al[365, 2] := 1.28657;
    fTable_Al[366, 0] := 3330.28; fTable_Al[366, 1] := 13.3973; fTable_Al[366, 2] := 1.25064;
    fTable_Al[367, 0] := 3384.15; fTable_Al[367, 1] := 13.4007; fTable_Al[367, 2] := 1.21564;
    fTable_Al[368, 0] := 3438.88; fTable_Al[368, 1] := 13.4034; fTable_Al[368, 2] := 1.18154;
    fTable_Al[369, 0] := 3494.50; fTable_Al[369, 1] := 13.4055; fTable_Al[369, 2] := 1.14831;
    fTable_Al[370, 0] := 3551.02; fTable_Al[370, 1] := 13.4070; fTable_Al[370, 2] := 1.11591;
    fTable_Al[371, 0] := 3608.46; fTable_Al[371, 1] := 13.4080; fTable_Al[371, 2] := 1.08436;
    fTable_Al[372, 0] := 3666.82; fTable_Al[372, 1] := 13.4085; fTable_Al[372, 2] := 1.05363;
    fTable_Al[373, 0] := 3726.13; fTable_Al[373, 1] := 13.4085; fTable_Al[373, 2] := 1.02369;
    fTable_Al[374, 0] := 3786.40; fTable_Al[374, 1] := 13.4081; fTable_Al[374, 2] := 0.994542;
    fTable_Al[375, 0] := 3847.64; fTable_Al[375, 1] := 13.4072; fTable_Al[375, 2] := 0.966167;
    fTable_Al[376, 0] := 3909.87; fTable_Al[376, 1] := 13.4060; fTable_Al[376, 2] := 0.938535;
    fTable_Al[377, 0] := 3973.11; fTable_Al[377, 1] := 13.4044; fTable_Al[377, 2] := 0.911645;
    fTable_Al[378, 0] := 4037.38; fTable_Al[378, 1] := 13.4025; fTable_Al[378, 2] := 0.885448;
    fTable_Al[379, 0] := 4102.68; fTable_Al[379, 1] := 13.4003; fTable_Al[379, 2] := 0.859966;
    fTable_Al[380, 0] := 4169.03; fTable_Al[380, 1] := 13.3978; fTable_Al[380, 2] := 0.835163;
    fTable_Al[381, 0] := 4236.46; fTable_Al[381, 1] := 13.3950; fTable_Al[381, 2] := 0.811033;
    fTable_Al[382, 0] := 4304.98; fTable_Al[382, 1] := 13.3920; fTable_Al[382, 2] := 0.787559;
    fTable_Al[383, 0] := 4374.62; fTable_Al[383, 1] := 13.3888; fTable_Al[383, 2] := 0.764708;
    fTable_Al[384, 0] := 4445.37; fTable_Al[384, 1] := 13.3853; fTable_Al[384, 2] := 0.742491;
    fTable_Al[385, 0] := 4517.27; fTable_Al[385, 1] := 13.3817; fTable_Al[385, 2] := 0.720878;
    fTable_Al[386, 0] := 4590.33; fTable_Al[386, 1] := 13.3779; fTable_Al[386, 2] := 0.699839;
    fTable_Al[387, 0] := 4664.58; fTable_Al[387, 1] := 13.3739; fTable_Al[387, 2] := 0.679399;
    fTable_Al[388, 0] := 4740.03; fTable_Al[388, 1] := 13.3698; fTable_Al[388, 2] := 0.659516;
    fTable_Al[389, 0] := 4816.69; fTable_Al[389, 1] := 13.3656; fTable_Al[389, 2] := 0.640176;
    fTable_Al[390, 0] := 4894.60; fTable_Al[390, 1] := 13.3612; fTable_Al[390, 2] := 0.621389;
    fTable_Al[391, 0] := 4973.77; fTable_Al[391, 1] := 13.3568; fTable_Al[391, 2] := 0.603106;
    fTable_Al[392, 0] := 5054.21; fTable_Al[392, 1] := 13.3522; fTable_Al[392, 2] := 0.585342;
    fTable_Al[393, 0] := 5135.96; fTable_Al[393, 1] := 13.3476; fTable_Al[393, 2] := 0.568080;
    fTable_Al[394, 0] := 5219.03; fTable_Al[394, 1] := 13.3429; fTable_Al[394, 2] := 0.551279;
    fTable_Al[395, 0] := 5303.44; fTable_Al[395, 1] := 13.3381; fTable_Al[395, 2] := 0.534968;
    fTable_Al[396, 0] := 5389.22; fTable_Al[396, 1] := 13.3332; fTable_Al[396, 2] := 0.519116;
    fTable_Al[397, 0] := 5476.39; fTable_Al[397, 1] := 13.3284; fTable_Al[397, 2] := 0.503715;
    fTable_Al[398, 0] := 5564.97; fTable_Al[398, 1] := 13.3235; fTable_Al[398, 2] := 0.488726;
    fTable_Al[399, 0] := 5654.98; fTable_Al[399, 1] := 13.3185; fTable_Al[399, 2] := 0.474187;
    fTable_Al[400, 0] := 5746.44; fTable_Al[400, 1] := 13.3135; fTable_Al[400, 2] := 0.460062;
    fTable_Al[401, 0] := 5839.39; fTable_Al[401, 1] := 13.3086; fTable_Al[401, 2] := 0.446336;
    fTable_Al[402, 0] := 5933.83; fTable_Al[402, 1] := 13.3036; fTable_Al[402, 2] := 0.433003;
    fTable_Al[403, 0] := 6029.81; fTable_Al[403, 1] := 13.2986; fTable_Al[403, 2] := 0.420026;
    fTable_Al[404, 0] := 6127.33; fTable_Al[404, 1] := 13.2936; fTable_Al[404, 2] := 0.407459;
    fTable_Al[405, 0] := 6226.44; fTable_Al[405, 1] := 13.2886; fTable_Al[405, 2] := 0.395224;
    fTable_Al[406, 0] := 6327.15; fTable_Al[406, 1] := 13.2836; fTable_Al[406, 2] := 0.383348;
    fTable_Al[407, 0] := 6429.48; fTable_Al[407, 1] := 13.2786; fTable_Al[407, 2] := 0.371815;
    fTable_Al[408, 0] := 6533.48; fTable_Al[408, 1] := 13.2737; fTable_Al[408, 2] := 0.360616;
    fTable_Al[409, 0] := 6639.15; fTable_Al[409, 1] := 13.2687; fTable_Al[409, 2] := 0.349739;
    fTable_Al[410, 0] := 6746.54; fTable_Al[410, 1] := 13.2638; fTable_Al[410, 2] := 0.339182;
    fTable_Al[411, 0] := 6855.65; fTable_Al[411, 1] := 13.2590; fTable_Al[411, 2] := 0.328927;
    fTable_Al[412, 0] := 6966.54; fTable_Al[412, 1] := 13.2541; fTable_Al[412, 2] := 0.318973;
    fTable_Al[413, 0] := 7079.22; fTable_Al[413, 1] := 13.2493; fTable_Al[413, 2] := 0.309309;
    fTable_Al[414, 0] := 7193.72; fTable_Al[414, 1] := 13.2446; fTable_Al[414, 2] := 0.299926;
    fTable_Al[415, 0] := 7310.07; fTable_Al[415, 1] := 13.2398; fTable_Al[415, 2] := 0.290817;
    fTable_Al[416, 0] := 7428.31; fTable_Al[416, 1] := 13.2352; fTable_Al[416, 2] := 0.281974;
    fTable_Al[417, 0] := 7548.45; fTable_Al[417, 1] := 13.2305; fTable_Al[417, 2] := 0.273391;
    fTable_Al[418, 0] := 7670.54; fTable_Al[418, 1] := 13.2259; fTable_Al[418, 2] := 0.265058;
    fTable_Al[419, 0] := 7794.61; fTable_Al[419, 1] := 13.2214; fTable_Al[419, 2] := 0.256972;
    fTable_Al[420, 0] := 7920.68; fTable_Al[420, 1] := 13.2169; fTable_Al[420, 2] := 0.249121;
    fTable_Al[421, 0] := 8048.79; fTable_Al[421, 1] := 13.2124; fTable_Al[421, 2] := 0.241506;
    fTable_Al[422, 0] := 8178.98; fTable_Al[422, 1] := 13.2081; fTable_Al[422, 2] := 0.234114;
    fTable_Al[423, 0] := 8311.26; fTable_Al[423, 1] := 13.2037; fTable_Al[423, 2] := 0.226938;
    fTable_Al[424, 0] := 8445.69; fTable_Al[424, 1] := 13.1994; fTable_Al[424, 2] := 0.219978;
    fTable_Al[425, 0] := 8582.29; fTable_Al[425, 1] := 13.1952; fTable_Al[425, 2] := 0.213218;
    fTable_Al[426, 0] := 8721.11; fTable_Al[426, 1] := 13.1910; fTable_Al[426, 2] := 0.206663;
    fTable_Al[427, 0] := 8862.16; fTable_Al[427, 1] := 13.1869; fTable_Al[427, 2] := 0.200304;
    fTable_Al[428, 0] := 9005.50; fTable_Al[428, 1] := 13.1829; fTable_Al[428, 2] := 0.194131;
    fTable_Al[429, 0] := 9151.16; fTable_Al[429, 1] := 13.1789; fTable_Al[429, 2] := 0.188140;
    fTable_Al[430, 0] := 9299.17; fTable_Al[430, 1] := 13.1749; fTable_Al[430, 2] := 0.182331;
    fTable_Al[431, 0] := 9449.58; fTable_Al[431, 1] := 13.1711; fTable_Al[431, 2] := 0.176693;
    fTable_Al[432, 0] := 9602.42; fTable_Al[432, 1] := 13.1672; fTable_Al[432, 2] := 0.171229;
    fTable_Al[433, 0] := 9757.73; fTable_Al[433, 1] := 13.1635; fTable_Al[433, 2] := 0.165921;
    fTable_Al[434, 0] := 9915.55; fTable_Al[434, 1] := 13.1598; fTable_Al[434, 2] := 0.160780;
    fTable_Al[435, 0] := 10075.9; fTable_Al[435, 1] := 13.1561; fTable_Al[435, 2] := 0.155788;
    fTable_Al[436, 0] := 10238.9; fTable_Al[436, 1] := 13.1526; fTable_Al[436, 2] := 0.150945;
    fTable_Al[437, 0] := 10404.5; fTable_Al[437, 1] := 13.1490; fTable_Al[437, 2] := 0.146248;
    fTable_Al[438, 0] := 10572.8; fTable_Al[438, 1] := 13.1456; fTable_Al[438, 2] := 0.141693;
    fTable_Al[439, 0] := 10743.8; fTable_Al[439, 1] := 13.1422; fTable_Al[439, 2] := 0.137274;
    fTable_Al[440, 0] := 10917.6; fTable_Al[440, 1] := 13.1388; fTable_Al[440, 2] := 0.132988;
    fTable_Al[441, 0] := 11094.2; fTable_Al[441, 1] := 13.1355; fTable_Al[441, 2] := 0.128831;
    fTable_Al[442, 0] := 11273.6; fTable_Al[442, 1] := 13.1323; fTable_Al[442, 2] := 0.124800;
    fTable_Al[443, 0] := 11455.9; fTable_Al[443, 1] := 13.1291; fTable_Al[443, 2] := 0.120890;
    fTable_Al[444, 0] := 11641.2; fTable_Al[444, 1] := 13.1260; fTable_Al[444, 2] := 0.117099;
    fTable_Al[445, 0] := 11829.5; fTable_Al[445, 1] := 13.1229; fTable_Al[445, 2] := 0.113422;
    fTable_Al[446, 0] := 12020.8; fTable_Al[446, 1] := 13.1199; fTable_Al[446, 2] := 0.109856;
    fTable_Al[447, 0] := 12215.3; fTable_Al[447, 1] := 13.1170; fTable_Al[447, 2] := 0.106398;
    fTable_Al[448, 0] := 12412.8; fTable_Al[448, 1] := 13.1141; fTable_Al[448, 2] := 0.103045;
    fTable_Al[449, 0] := 12613.6; fTable_Al[449, 1] := 13.1112; fTable_Al[449, 2] := 0.0997941;
    fTable_Al[450, 0] := 12817.6; fTable_Al[450, 1] := 13.1084; fTable_Al[450, 2] := 0.0966416;
    fTable_Al[451, 0] := 13025.0; fTable_Al[451, 1] := 13.1057; fTable_Al[451, 2] := 0.0935848;
    fTable_Al[452, 0] := 13235.6; fTable_Al[452, 1] := 13.1030; fTable_Al[452, 2] := 0.0906209;
    fTable_Al[453, 0] := 13449.7; fTable_Al[453, 1] := 13.1004; fTable_Al[453, 2] := 0.0877473;
    fTable_Al[454, 0] := 13667.2; fTable_Al[454, 1] := 13.0978; fTable_Al[454, 2] := 0.0849611;
    fTable_Al[455, 0] := 13888.3; fTable_Al[455, 1] := 13.0953; fTable_Al[455, 2] := 0.0822598;
    fTable_Al[456, 0] := 14112.9; fTable_Al[456, 1] := 13.0928; fTable_Al[456, 2] := 0.0796408;
    fTable_Al[457, 0] := 14341.2; fTable_Al[457, 1] := 13.0903; fTable_Al[457, 2] := 0.0771018;
    fTable_Al[458, 0] := 14573.1; fTable_Al[458, 1] := 13.0880; fTable_Al[458, 2] := 0.0746402;
    fTable_Al[459, 0] := 14808.9; fTable_Al[459, 1] := 13.0856; fTable_Al[459, 2] := 0.0722539;
    fTable_Al[460, 0] := 15048.4; fTable_Al[460, 1] := 13.0833; fTable_Al[460, 2] := 0.0699405;
    fTable_Al[461, 0] := 15291.8; fTable_Al[461, 1] := 13.0811; fTable_Al[461, 2] := 0.0676979;
    fTable_Al[462, 0] := 15539.1; fTable_Al[462, 1] := 13.0789; fTable_Al[462, 2] := 0.0655240;
    fTable_Al[463, 0] := 15790.4; fTable_Al[463, 1] := 13.0768; fTable_Al[463, 2] := 0.0634165;
    fTable_Al[464, 0] := 16045.8; fTable_Al[464, 1] := 13.0746; fTable_Al[464, 2] := 0.0613737;
    fTable_Al[465, 0] := 16305.4; fTable_Al[465, 1] := 13.0726; fTable_Al[465, 2] := 0.0593935;
    fTable_Al[466, 0] := 16569.1; fTable_Al[466, 1] := 13.0706; fTable_Al[466, 2] := 0.0574741;
    fTable_Al[467, 0] := 16837.1; fTable_Al[467, 1] := 13.0686; fTable_Al[467, 2] := 0.0556136;
    fTable_Al[468, 0] := 17109.4; fTable_Al[468, 1] := 13.0667; fTable_Al[468, 2] := 0.0538102;
    fTable_Al[469, 0] := 17386.1; fTable_Al[469, 1] := 13.0648; fTable_Al[469, 2] := 0.0520623;
    fTable_Al[470, 0] := 17667.4; fTable_Al[470, 1] := 13.0629; fTable_Al[470, 2] := 0.0503681;
    fTable_Al[471, 0] := 17953.1; fTable_Al[471, 1] := 13.0611; fTable_Al[471, 2] := 0.0487260;
    fTable_Al[472, 0] := 18243.5; fTable_Al[472, 1] := 13.0593; fTable_Al[472, 2] := 0.0471345;
    fTable_Al[473, 0] := 18538.6; fTable_Al[473, 1] := 13.0576; fTable_Al[473, 2] := 0.0455920;
    fTable_Al[474, 0] := 18838.4; fTable_Al[474, 1] := 13.0559; fTable_Al[474, 2] := 0.0440970;
    fTable_Al[475, 0] := 19143.1; fTable_Al[475, 1] := 13.0542; fTable_Al[475, 2] := 0.0426482;
    fTable_Al[476, 0] := 19452.7; fTable_Al[476, 1] := 13.0526; fTable_Al[476, 2] := 0.0412440;
    fTable_Al[477, 0] := 19767.4; fTable_Al[477, 1] := 13.0510; fTable_Al[477, 2] := 0.0398831;
    fTable_Al[478, 0] := 20087.1; fTable_Al[478, 1] := 13.0494; fTable_Al[478, 2] := 0.0385533;
    fTable_Al[479, 0] := 20412.0; fTable_Al[479, 1] := 13.0479; fTable_Al[479, 2] := 0.0372771;
    fTable_Al[480, 0] := 20742.1; fTable_Al[480, 1] := 13.0464; fTable_Al[480, 2] := 0.0360423;
    fTable_Al[481, 0] := 21077.6; fTable_Al[481, 1] := 13.0449; fTable_Al[481, 2] := 0.0348475;
    fTable_Al[482, 0] := 21418.5; fTable_Al[482, 1] := 13.0435; fTable_Al[482, 2] := 0.0336915;
    fTable_Al[483, 0] := 21765.0; fTable_Al[483, 1] := 13.0421; fTable_Al[483, 2] := 0.0325731;
    fTable_Al[484, 0] := 22117.0; fTable_Al[484, 1] := 13.0407; fTable_Al[484, 2] := 0.0314909;
    fTable_Al[485, 0] := 22474.7; fTable_Al[485, 1] := 13.0394; fTable_Al[485, 2] := 0.0304440;
    fTable_Al[486, 0] := 22838.2; fTable_Al[486, 1] := 13.0381; fTable_Al[486, 2] := 0.0294311;
    fTable_Al[487, 0] := 23207.6; fTable_Al[487, 1] := 13.0368; fTable_Al[487, 2] := 0.0284511;
    fTable_Al[488, 0] := 23583.0; fTable_Al[488, 1] := 13.0356; fTable_Al[488, 2] := 0.0275030;
    fTable_Al[489, 0] := 23964.4; fTable_Al[489, 1] := 13.0343; fTable_Al[489, 2] := 0.0265858;
    fTable_Al[490, 0] := 24352.0; fTable_Al[490, 1] := 13.0331; fTable_Al[490, 2] := 0.0256985;
    fTable_Al[491, 0] := 24745.9; fTable_Al[491, 1] := 13.0320; fTable_Al[491, 2] := 0.0248401;
    fTable_Al[492, 0] := 25146.2; fTable_Al[492, 1] := 13.0308; fTable_Al[492, 2] := 0.0240097;
    fTable_Al[493, 0] := 25552.9; fTable_Al[493, 1] := 13.0297; fTable_Al[493, 2] := 0.0232064;
    fTable_Al[494, 0] := 25966.2; fTable_Al[494, 1] := 13.0287; fTable_Al[494, 2] := 0.0224293;
    fTable_Al[495, 0] := 26386.1; fTable_Al[495, 1] := 13.0276; fTable_Al[495, 2] := 0.0216776;
    fTable_Al[496, 0] := 26812.9; fTable_Al[496, 1] := 13.0266; fTable_Al[496, 2] := 0.0209505;
    fTable_Al[497, 0] := 27246.6; fTable_Al[497, 1] := 13.0256; fTable_Al[497, 2] := 0.0202471;
    fTable_Al[498, 0] := 27687.3; fTable_Al[498, 1] := 13.0246; fTable_Al[498, 2] := 0.0195668;
    fTable_Al[499, 0] := 28135.1; fTable_Al[499, 1] := 13.0236; fTable_Al[499, 2] := 0.0189087;
    fTable_Al[500, 0] := 28590.2; fTable_Al[500, 1] := 13.0227; fTable_Al[500, 2] := 0.0182722;
    fTable_Al[501, 0] := 29052.6; fTable_Al[501, 1] := 13.0218; fTable_Al[501, 2] := 0.0176565;
    fTable_Al[502, 0] := 29522.5; fTable_Al[502, 1] := 13.0209; fTable_Al[502, 2] := 0.0170611;
    fTable_Al[503, 0] := 30000.0; fTable_Al[503, 1] := 13.0198; fTable_Al[503, 2] := 0.0164852;

    (* Table initialization: fTable_Be *)
    fTable_Be[0, 0] := 10.0000; fTable_Be[0, 1] := -9999; fTable_Be[0, 2] := 1.70333;
    fTable_Be[1, 0] := 10.1617; fTable_Be[1, 1] := -9999; fTable_Be[1, 2] := 1.71802;
    fTable_Be[2, 0] := 10.3261; fTable_Be[2, 1] := -9999; fTable_Be[2, 2] := 1.73284;
    fTable_Be[3, 0] := 10.4931; fTable_Be[3, 1] := -9999; fTable_Be[3, 2] := 1.74778;
    fTable_Be[4, 0] := 10.6628; fTable_Be[4, 1] := -9999; fTable_Be[4, 2] := 1.75737;
    fTable_Be[5, 0] := 10.8353; fTable_Be[5, 1] := -9999; fTable_Be[5, 2] := 1.76678;
    fTable_Be[6, 0] := 11.0105; fTable_Be[6, 1] := -9999; fTable_Be[6, 2] := 1.77624;
    fTable_Be[7, 0] := 11.1886; fTable_Be[7, 1] := -9999; fTable_Be[7, 2] := 1.78574;
    fTable_Be[8, 0] := 11.3696; fTable_Be[8, 1] := -9999; fTable_Be[8, 2] := 1.79530;
    fTable_Be[9, 0] := 11.5535; fTable_Be[9, 1] := -9999; fTable_Be[9, 2] := 1.80306;
    fTable_Be[10, 0] := 11.7404; fTable_Be[10, 1] := -9999; fTable_Be[10, 2] := 1.80629;
    fTable_Be[11, 0] := 11.9303; fTable_Be[11, 1] := -9999; fTable_Be[11, 2] := 1.80952;
    fTable_Be[12, 0] := 12.1232; fTable_Be[12, 1] := -9999; fTable_Be[12, 2] := 1.81276;
    fTable_Be[13, 0] := 12.3193; fTable_Be[13, 1] := -9999; fTable_Be[13, 2] := 1.81600;
    fTable_Be[14, 0] := 12.5186; fTable_Be[14, 1] := -9999; fTable_Be[14, 2] := 1.81871;
    fTable_Be[15, 0] := 12.7210; fTable_Be[15, 1] := -9999; fTable_Be[15, 2] := 1.81609;
    fTable_Be[16, 0] := 12.9268; fTable_Be[16, 1] := -9999; fTable_Be[16, 2] := 1.81347;
    fTable_Be[17, 0] := 13.1359; fTable_Be[17, 1] := -9999; fTable_Be[17, 2] := 1.80922;
    fTable_Be[18, 0] := 13.3483; fTable_Be[18, 1] := -9999; fTable_Be[18, 2] := 1.80410;
    fTable_Be[19, 0] := 13.5642; fTable_Be[19, 1] := -9999; fTable_Be[19, 2] := 1.79747;
    fTable_Be[20, 0] := 13.7836; fTable_Be[20, 1] := -9999; fTable_Be[20, 2] := 1.78729;
    fTable_Be[21, 0] := 14.0066; fTable_Be[21, 1] := -9999; fTable_Be[21, 2] := 1.77705;
    fTable_Be[22, 0] := 14.2331; fTable_Be[22, 1] := -9999; fTable_Be[22, 2] := 1.76267;
    fTable_Be[23, 0] := 14.4633; fTable_Be[23, 1] := -9999; fTable_Be[23, 2] := 1.74841;
    fTable_Be[24, 0] := 14.6972; fTable_Be[24, 1] := -9999; fTable_Be[24, 2] := 1.72956;
    fTable_Be[25, 0] := 14.9350; fTable_Be[25, 1] := -9999; fTable_Be[25, 2] := 1.71004;
    fTable_Be[26, 0] := 15.1765; fTable_Be[26, 1] := -9999; fTable_Be[26, 2] := 1.68541;
    fTable_Be[27, 0] := 15.4220; fTable_Be[27, 1] := -9999; fTable_Be[27, 2] := 1.65917;
    fTable_Be[28, 0] := 15.6714; fTable_Be[28, 1] := -9999; fTable_Be[28, 2] := 1.62778;
    fTable_Be[29, 0] := 15.9249; fTable_Be[29, 1] := -9999; fTable_Be[29, 2] := 1.59448;
    fTable_Be[30, 0] := 16.1825; fTable_Be[30, 1] := -9999; fTable_Be[30, 2] := 1.55788;
    fTable_Be[31, 0] := 16.4442; fTable_Be[31, 1] := -9999; fTable_Be[31, 2] := 1.52050;
    fTable_Be[32, 0] := 16.7102; fTable_Be[32, 1] := -9999; fTable_Be[32, 2] := 1.47675;
    fTable_Be[33, 0] := 16.9805; fTable_Be[33, 1] := -9999; fTable_Be[33, 2] := 1.43237;
    fTable_Be[34, 0] := 17.2551; fTable_Be[34, 1] := -9999; fTable_Be[34, 2] := 1.38176;
    fTable_Be[35, 0] := 17.5342; fTable_Be[35, 1] := -9999; fTable_Be[35, 2] := 1.33102;
    fTable_Be[36, 0] := 17.8178; fTable_Be[36, 1] := -9999; fTable_Be[36, 2] := 1.27265;
    fTable_Be[37, 0] := 18.1060; fTable_Be[37, 1] := -9999; fTable_Be[37, 2] := 1.22588;
    fTable_Be[38, 0] := 18.3988; fTable_Be[38, 1] := -9999; fTable_Be[38, 2] := 1.19605;
    fTable_Be[39, 0] := 18.6964; fTable_Be[39, 1] := -9999; fTable_Be[39, 2] := 1.16961;
    fTable_Be[40, 0] := 18.9988; fTable_Be[40, 1] := -9999; fTable_Be[40, 2] := 1.14509;
    fTable_Be[41, 0] := 19.3061; fTable_Be[41, 1] := 2.30967; fTable_Be[41, 2] := 1.10518;
    fTable_Be[42, 0] := 19.6184; fTable_Be[42, 1] := 2.31367; fTable_Be[42, 2] := 1.06950;
    fTable_Be[43, 0] := 19.9357; fTable_Be[43, 1] := 2.31537; fTable_Be[43, 2] := 1.03964;
    fTable_Be[44, 0] := 20.2581; fTable_Be[44, 1] := 2.31755; fTable_Be[44, 2] := 1.01722;
    fTable_Be[45, 0] := 20.5858; fTable_Be[45, 1] := 2.32374; fTable_Be[45, 2] := 0.999039;
    fTable_Be[46, 0] := 20.9187; fTable_Be[46, 1] := 2.34045; fTable_Be[46, 2] := 0.987135;
    fTable_Be[47, 0] := 21.2571; fTable_Be[47, 1] := 2.37239; fTable_Be[47, 2] := 0.952742;
    fTable_Be[48, 0] := 21.6009; fTable_Be[48, 1] := 2.38699; fTable_Be[48, 2] := 0.912693;
    fTable_Be[49, 0] := 21.9503; fTable_Be[49, 1] := 2.39600; fTable_Be[49, 2] := 0.874329;
    fTable_Be[50, 0] := 22.3053; fTable_Be[50, 1] := 2.40177; fTable_Be[50, 2] := 0.837576;
    fTable_Be[51, 0] := 22.6661; fTable_Be[51, 1] := 2.40538; fTable_Be[51, 2] := 0.802368;
    fTable_Be[52, 0] := 23.0327; fTable_Be[52, 1] := 2.40746; fTable_Be[52, 2] := 0.768641;
    fTable_Be[53, 0] := 23.4052; fTable_Be[53, 1] := 2.40846; fTable_Be[53, 2] := 0.736331;
    fTable_Be[54, 0] := 23.7838; fTable_Be[54, 1] := 2.40939; fTable_Be[54, 2] := 0.705380;
    fTable_Be[55, 0] := 24.1685; fTable_Be[55, 1] := 2.41248; fTable_Be[55, 2] := 0.675729;
    fTable_Be[56, 0] := 24.5594; fTable_Be[56, 1] := 2.41570; fTable_Be[56, 2] := 0.647325;
    fTable_Be[57, 0] := 24.9566; fTable_Be[57, 1] := 2.42027; fTable_Be[57, 2] := 0.609275;
    fTable_Be[58, 0] := 25.3602; fTable_Be[58, 1] := 2.41808; fTable_Be[58, 2] := 0.567900;
    fTable_Be[59, 0] := 25.7704; fTable_Be[59, 1] := 2.40985; fTable_Be[59, 2] := 0.529334;
    fTable_Be[60, 0] := 26.1872; fTable_Be[60, 1] := 2.39826; fTable_Be[60, 2] := 0.493388;
    fTable_Be[61, 0] := 26.6108; fTable_Be[61, 1] := 2.38435; fTable_Be[61, 2] := 0.459883;
    fTable_Be[62, 0] := 27.0412; fTable_Be[62, 1] := 2.36859; fTable_Be[62, 2] := 0.428653;
    fTable_Be[63, 0] := 27.4786; fTable_Be[63, 1] := 2.35116; fTable_Be[63, 2] := 0.399544;
    fTable_Be[64, 0] := 27.9230; fTable_Be[64, 1] := 2.33226; fTable_Be[64, 2] := 0.372411;
    fTable_Be[65, 0] := 28.3747; fTable_Be[65, 1] := 2.30996; fTable_Be[65, 2] := 0.347121;
    fTable_Be[66, 0] := 28.8336; fTable_Be[66, 1] := 2.28594; fTable_Be[66, 2] := 0.328404;
    fTable_Be[67, 0] := 29.3000; fTable_Be[67, 1] := 2.26312; fTable_Be[67, 2] := 0.315229;
    fTable_Be[68, 0] := 29.7739; fTable_Be[68, 1] := 2.24541; fTable_Be[68, 2] := 0.302582;
    fTable_Be[69, 0] := 30.2554; fTable_Be[69, 1] := 2.22901; fTable_Be[69, 2] := 0.290443;
    fTable_Be[70, 0] := 30.7448; fTable_Be[70, 1] := 2.21325; fTable_Be[70, 2] := 0.278791;
    fTable_Be[71, 0] := 31.2421; fTable_Be[71, 1] := 2.19800; fTable_Be[71, 2] := 0.267606;
    fTable_Be[72, 0] := 31.7474; fTable_Be[72, 1] := 2.18311; fTable_Be[72, 2] := 0.256870;
    fTable_Be[73, 0] := 32.2609; fTable_Be[73, 1] := 2.16844; fTable_Be[73, 2] := 0.246565;
    fTable_Be[74, 0] := 32.7827; fTable_Be[74, 1] := 2.15391; fTable_Be[74, 2] := 0.236673;
    fTable_Be[75, 0] := 33.3129; fTable_Be[75, 1] := 2.13952; fTable_Be[75, 2] := 0.227178;
    fTable_Be[76, 0] := 33.8517; fTable_Be[76, 1] := 2.12325; fTable_Be[76, 2] := 0.218064;
    fTable_Be[77, 0] := 34.3992; fTable_Be[77, 1] := 2.10677; fTable_Be[77, 2] := 0.211374;
    fTable_Be[78, 0] := 34.9556; fTable_Be[78, 1] := 2.09142; fTable_Be[78, 2] := 0.206573;
    fTable_Be[79, 0] := 35.5210; fTable_Be[79, 1] := 2.07852; fTable_Be[79, 2] := 0.201882;
    fTable_Be[80, 0] := 36.0955; fTable_Be[80, 1] := 2.06586; fTable_Be[80, 2] := 0.197297;
    fTable_Be[81, 0] := 36.6793; fTable_Be[81, 1] := 2.05353; fTable_Be[81, 2] := 0.192816;
    fTable_Be[82, 0] := 37.2726; fTable_Be[82, 1] := 2.04141; fTable_Be[82, 2] := 0.188437;
    fTable_Be[83, 0] := 37.8754; fTable_Be[83, 1] := 2.02931; fTable_Be[83, 2] := 0.184157;
    fTable_Be[84, 0] := 38.4880; fTable_Be[84, 1] := 2.01697; fTable_Be[84, 2] := 0.179975;
    fTable_Be[85, 0] := 38.9000; fTable_Be[85, 1] := 2.00799; fTable_Be[85, 2] := 0.177252;
    fTable_Be[86, 0] := 39.2000; fTable_Be[86, 1] := 2.00121; fTable_Be[86, 2] := 0.176713;
    fTable_Be[87, 0] := 39.5000; fTable_Be[87, 1] := 1.99567; fTable_Be[87, 2] := 0.176983;
    fTable_Be[88, 0] := 39.9000; fTable_Be[88, 1] := 1.98913; fTable_Be[88, 2] := 0.175827;
    fTable_Be[89, 0] := 40.0000; fTable_Be[89, 1] := 1.98733; fTable_Be[89, 2] := 0.175565;
    fTable_Be[90, 0] := 40.2760; fTable_Be[90, 1] := 1.98264; fTable_Be[90, 2] := 0.174663;
    fTable_Be[91, 0] := 40.5560; fTable_Be[91, 1] := 1.97786; fTable_Be[91, 2] := 0.174609;
    fTable_Be[92, 0] := 40.6970; fTable_Be[92, 1] := 1.97610; fTable_Be[92, 2] := 0.174013;
    fTable_Be[93, 0] := 41.1270; fTable_Be[93, 1] := 1.96960; fTable_Be[93, 2] := 0.173456;
    fTable_Be[94, 0] := 41.5660; fTable_Be[94, 1] := 1.96327; fTable_Be[94, 2] := 0.171435;
    fTable_Be[95, 0] := 42.1670; fTable_Be[95, 1] := 1.95400; fTable_Be[95, 2] := 0.170039;
    fTable_Be[96, 0] := 42.4730; fTable_Be[96, 1] := 1.94966; fTable_Be[96, 2] := 0.168799;
    fTable_Be[97, 0] := 42.9420; fTable_Be[97, 1] := 1.94280; fTable_Be[97, 2] := 0.168198;
    fTable_Be[98, 0] := 43.2600; fTable_Be[98, 1] := 1.93854; fTable_Be[98, 2] := 0.166905;
    fTable_Be[99, 0] := 43.7460; fTable_Be[99, 1] := 1.93138; fTable_Be[99, 2] := 0.165791;
    fTable_Be[100, 0] := 44.0760; fTable_Be[100, 1] := 1.92708; fTable_Be[100, 2] := 0.165390;
    fTable_Be[101, 0] := 44.4110; fTable_Be[101, 1] := 1.92291; fTable_Be[101, 2] := 0.164383;
    fTable_Be[102, 0] := 44.5810; fTable_Be[102, 1] := 1.92070; fTable_Be[102, 2] := 0.163618;
    fTable_Be[103, 0] := 44.9240; fTable_Be[103, 1] := 1.91607; fTable_Be[103, 2] := 0.162962;
    fTable_Be[104, 0] := 45.2720; fTable_Be[104, 1] := 1.91126; fTable_Be[104, 2] := 0.161326;
    fTable_Be[105, 0] := 45.4480; fTable_Be[105, 1] := 1.90903; fTable_Be[105, 2] := 0.161038;
    fTable_Be[106, 0] := 45.9850; fTable_Be[106, 1] := 1.90129; fTable_Be[106, 2] := 0.159149;
    fTable_Be[107, 0] := 46.7288; fTable_Be[107, 1] := 1.89036; fTable_Be[107, 2] := 0.157516;
    fTable_Be[108, 0] := 47.4846; fTable_Be[108, 1] := 1.87948; fTable_Be[108, 2] := 0.155990;
    fTable_Be[109, 0] := 47.6740; fTable_Be[109, 1] := 1.87667; fTable_Be[109, 2] := 0.155621;
    fTable_Be[110, 0] := 48.2650; fTable_Be[110, 1] := 1.86782; fTable_Be[110, 2] := 0.155028;
    fTable_Be[111, 0] := 48.8710; fTable_Be[111, 1] := 1.85943; fTable_Be[111, 2] := 0.155666;
    fTable_Be[112, 0] := 49.0760; fTable_Be[112, 1] := 1.85755; fTable_Be[112, 2] := 0.155951;
    fTable_Be[113, 0] := 49.2830; fTable_Be[113, 1] := 1.85503; fTable_Be[113, 2] := 0.154508;
    fTable_Be[114, 0] := 49.8930; fTable_Be[114, 1] := 1.84657; fTable_Be[114, 2] := 0.154198;
    fTable_Be[115, 0] := 50.7000; fTable_Be[115, 1] := 1.83364; fTable_Be[115, 2] := 0.155814;
    fTable_Be[116, 0] := 51.5200; fTable_Be[116, 1] := 1.82367; fTable_Be[116, 2] := 0.157447;
    fTable_Be[117, 0] := 51.9010; fTable_Be[117, 1] := 1.81956; fTable_Be[117, 2] := 0.158203;
    fTable_Be[118, 0] := 52.4010; fTable_Be[118, 1] := 1.81434; fTable_Be[118, 2] := 0.158683;
    fTable_Be[119, 0] := 53.2485; fTable_Be[119, 1] := 1.80585; fTable_Be[119, 2] := 0.158768;
    fTable_Be[120, 0] := 53.4010; fTable_Be[120, 1] := 1.80449; fTable_Be[120, 2] := 0.158784;
    fTable_Be[121, 0] := 53.9000; fTable_Be[121, 1] := 1.79914; fTable_Be[121, 2] := 0.157647;
    fTable_Be[122, 0] := 54.4010; fTable_Be[122, 1] := 1.79325; fTable_Be[122, 2] := 0.156933;
    fTable_Be[123, 0] := 54.9010; fTable_Be[123, 1] := 1.78748; fTable_Be[123, 2] := 0.157035;
    fTable_Be[124, 0] := 55.4000; fTable_Be[124, 1] := 1.78219; fTable_Be[124, 2] := 0.156125;
    fTable_Be[125, 0] := 55.9010; fTable_Be[125, 1] := 1.77644; fTable_Be[125, 2] := 0.155633;
    fTable_Be[126, 0] := 56.8052; fTable_Be[126, 1] := 1.76616; fTable_Be[126, 2] := 0.152967;
    fTable_Be[127, 0] := 56.9010; fTable_Be[127, 1] := 1.76491; fTable_Be[127, 2] := 0.152689;
    fTable_Be[128, 0] := 57.4010; fTable_Be[128, 1] := 1.75779; fTable_Be[128, 2] := 0.151560;
    fTable_Be[129, 0] := 57.9010; fTable_Be[129, 1] := 1.75138; fTable_Be[129, 2] := 0.151256;
    fTable_Be[130, 0] := 58.4000; fTable_Be[130, 1] := 1.74467; fTable_Be[130, 2] := 0.149795;
    fTable_Be[131, 0] := 59.3446; fTable_Be[131, 1] := 1.73066; fTable_Be[131, 2] := 0.148143;
    fTable_Be[132, 0] := 60.3044; fTable_Be[132, 1] := 1.71666; fTable_Be[132, 2] := 0.147555;
    fTable_Be[133, 0] := 60.9010; fTable_Be[133, 1] := 1.70803; fTable_Be[133, 2] := 0.147236;
    fTable_Be[134, 0] := 61.4010; fTable_Be[134, 1] := 1.70036; fTable_Be[134, 2] := 0.146656;
    fTable_Be[135, 0] := 62.3941; fTable_Be[135, 1] := 1.68542; fTable_Be[135, 2] := 0.147197;
    fTable_Be[136, 0] := 62.4010; fTable_Be[136, 1] := 1.68532; fTable_Be[136, 2] := 0.147201;
    fTable_Be[137, 0] := 63.4000; fTable_Be[137, 1] := 1.67044; fTable_Be[137, 2] := 0.146706;
    fTable_Be[138, 0] := 63.9020; fTable_Be[138, 1] := 1.66247; fTable_Be[138, 2] := 0.147388;
    fTable_Be[139, 0] := 64.4000; fTable_Be[139, 1] := 1.65492; fTable_Be[139, 2] := 0.147185;
    fTable_Be[140, 0] := 65.4010; fTable_Be[140, 1] := 1.63983; fTable_Be[140, 2] := 0.147806;
    fTable_Be[141, 0] := 65.9010; fTable_Be[141, 1] := 1.63182; fTable_Be[141, 2] := 0.147426;
    fTable_Be[142, 0] := 66.9669; fTable_Be[142, 1] := 1.61497; fTable_Be[142, 2] := 0.147801;
    fTable_Be[143, 0] := 68.0500; fTable_Be[143, 1] := 1.59766; fTable_Be[143, 2] := 0.147747;
    fTable_Be[144, 0] := 69.1507; fTable_Be[144, 1] := 1.57948; fTable_Be[144, 2] := 0.147404;
    fTable_Be[145, 0] := 69.4010; fTable_Be[145, 1] := 1.57524; fTable_Be[145, 2] := 0.147327;
    fTable_Be[146, 0] := 70.2340; fTable_Be[146, 1] := 1.56001; fTable_Be[146, 2] := 0.145950;
    fTable_Be[147, 0] := 71.3700; fTable_Be[147, 1] := 1.53888; fTable_Be[147, 2] := 0.145981;
    fTable_Be[148, 0] := 72.5243; fTable_Be[148, 1] := 1.51676; fTable_Be[148, 2] := 0.146011;
    fTable_Be[149, 0] := 72.5670; fTable_Be[149, 1] := 1.51586; fTable_Be[149, 2] := 0.146012;
    fTable_Be[150, 0] := 72.9000; fTable_Be[150, 1] := 1.50929; fTable_Be[150, 2] := 0.145632;
    fTable_Be[151, 0] := 73.5680; fTable_Be[151, 1] := 1.49567; fTable_Be[151, 2] := 0.146079;
    fTable_Be[152, 0] := 74.7579; fTable_Be[152, 1] := 1.47049; fTable_Be[152, 2] := 0.146106;
    fTable_Be[153, 0] := 74.9000; fTable_Be[153, 1] := 1.46741; fTable_Be[153, 2] := 0.146109;
    fTable_Be[154, 0] := 75.2350; fTable_Be[154, 1] := 1.46015; fTable_Be[154, 2] := 0.146426;
    fTable_Be[155, 0] := 75.5670; fTable_Be[155, 1] := 1.45305; fTable_Be[155, 2] := 0.146447;
    fTable_Be[156, 0] := 76.5680; fTable_Be[156, 1] := 1.43052; fTable_Be[156, 2] := 0.147310;
    fTable_Be[157, 0] := 77.2350; fTable_Be[157, 1] := 1.41539; fTable_Be[157, 2] := 0.147639;
    fTable_Be[158, 0] := 77.5670; fTable_Be[158, 1] := 1.40764; fTable_Be[158, 2] := 0.148124;
    fTable_Be[159, 0] := 77.9010; fTable_Be[159, 1] := 1.40006; fTable_Be[159, 2] := 0.148179;
    fTable_Be[160, 0] := 78.5670; fTable_Be[160, 1] := 1.38396; fTable_Be[160, 2] := 0.148938;
    fTable_Be[161, 0] := 78.9000; fTable_Be[161, 1] := 1.37631; fTable_Be[161, 2] := 0.148969;
    fTable_Be[162, 0] := 80.1761; fTable_Be[162, 1] := 1.34408; fTable_Be[162, 2] := 0.150222;
    fTable_Be[163, 0] := 80.9000; fTable_Be[163, 1] := 1.32524; fTable_Be[163, 2] := 0.150928;
    fTable_Be[164, 0] := 81.2340; fTable_Be[164, 1] := 1.31669; fTable_Be[164, 2] := 0.151099;
    fTable_Be[165, 0] := 81.5680; fTable_Be[165, 1] := 1.30817; fTable_Be[165, 2] := 0.151573;
    fTable_Be[166, 0] := 82.8873; fTable_Be[166, 1] := 1.27205; fTable_Be[166, 2] := 0.152380;
    fTable_Be[167, 0] := 83.5680; fTable_Be[167, 1] := 1.25273; fTable_Be[167, 2] := 0.152793;
    fTable_Be[168, 0] := 84.9010; fTable_Be[168, 1] := 1.21283; fTable_Be[168, 2] := 0.152919;
    fTable_Be[169, 0] := 86.2742; fTable_Be[169, 1] := 1.16875; fTable_Be[169, 2] := 0.153088;
    fTable_Be[170, 0] := 87.6696; fTable_Be[170, 1] := 1.12068; fTable_Be[170, 2] := 0.152944;
    fTable_Be[171, 0] := 89.0876; fTable_Be[171, 1] := 1.06780; fTable_Be[171, 2] := 0.152717;
    fTable_Be[172, 0] := 90.5285; fTable_Be[172, 1] := 1.00938; fTable_Be[172, 2] := 0.152457;
    fTable_Be[173, 0] := 91.9928; fTable_Be[173, 1] := 0.944630; fTable_Be[173, 2] := 0.152189;
    fTable_Be[174, 0] := 93.4807; fTable_Be[174, 1] := 0.872376; fTable_Be[174, 2] := 0.151920;
    fTable_Be[175, 0] := 94.9926; fTable_Be[175, 1] := 0.791324; fTable_Be[175, 2] := 0.151867;
    fTable_Be[176, 0] := 96.5291; fTable_Be[176, 1] := 0.699761; fTable_Be[176, 2] := 0.151828;
    fTable_Be[177, 0] := 97.5670; fTable_Be[177, 1] := 0.631310; fTable_Be[177, 2] := 0.151801;
    fTable_Be[178, 0] := 98.5680; fTable_Be[178, 1] := 0.560328; fTable_Be[178, 2] := 0.152508;
    fTable_Be[179, 0] := 98.7770; fTable_Be[179, 1] := 0.544993; fTable_Be[179, 2] := 0.152245;
    fTable_Be[180, 0] := 99.5260; fTable_Be[180, 1] := 0.486543; fTable_Be[180, 2] := 0.151861;
    fTable_Be[181, 0] := 99.9010; fTable_Be[181, 1] := 0.455599; fTable_Be[181, 2] := 0.151904;
    fTable_Be[182, 0] := 100.270; fTable_Be[182, 1] := 0.424344; fTable_Be[182, 2] := 0.151744;
    fTable_Be[183, 0] := 100.660; fTable_Be[183, 1] := 0.389731; fTable_Be[183, 2] := 0.152054;
    fTable_Be[184, 0] := 102.030; fTable_Be[184, 1] := 0.258588; fTable_Be[184, 2] := 0.151656;
    fTable_Be[185, 0] := 102.400; fTable_Be[185, 1] := 0.219148; fTable_Be[185, 2] := 0.151818;
    fTable_Be[186, 0] := 103.770; fTable_Be[186, 1] := 0.0597848; fTable_Be[186, 2] := 0.151969;
    fTable_Be[187, 0] := 104.030; fTable_Be[187, 1] := 0.0260858; fTable_Be[187, 2] := 0.152169;
    fTable_Be[188, 0] := 105.530; fTable_Be[188, 1] := -0.191568; fTable_Be[188, 2] := 0.151371;
    fTable_Be[189, 0] := 106.530; fTable_Be[189, 1] := -0.368308; fTable_Be[189, 2] := 0.151676;
    fTable_Be[190, 0] := 106.900; fTable_Be[190, 1] := -0.441904; fTable_Be[190, 2] := 0.152246;
    fTable_Be[191, 0] := 107.770; fTable_Be[191, 1] := -0.637412; fTable_Be[191, 2] := 0.154099;
    fTable_Be[192, 0] := 108.030; fTable_Be[192, 1] := -0.702374; fTable_Be[192, 2] := 0.155662;
    fTable_Be[193, 0] := 108.280; fTable_Be[193, 1] := -0.768299; fTable_Be[193, 2] := 0.156220;
    fTable_Be[194, 0] := 108.400; fTable_Be[194, 1] := -0.802126; fTable_Be[194, 2] := 0.155741;
    fTable_Be[195, 0] := 108.530; fTable_Be[195, 1] := -0.840651; fTable_Be[195, 2] := 0.156004;
    fTable_Be[196, 0] := 108.650; fTable_Be[196, 1] := -0.876311; fTable_Be[196, 2] := 0.158215;
    fTable_Be[197, 0] := 108.770; fTable_Be[197, 1] := -0.912731; fTable_Be[197, 2] := 0.158122;
    fTable_Be[198, 0] := 109.030; fTable_Be[198, 1] := -0.997553; fTable_Be[198, 2] := 0.159793;
    fTable_Be[199, 0] := 109.150; fTable_Be[199, 1] := -1.03849; fTable_Be[199, 2] := 0.161052;
    fTable_Be[200, 0] := 109.270; fTable_Be[200, 1] := -1.08113; fTable_Be[200, 2] := 0.161306;
    fTable_Be[201, 0] := 109.400; fTable_Be[201, 1] := -1.12894; fTable_Be[201, 2] := 0.163454;
    fTable_Be[202, 0] := 109.530; fTable_Be[202, 1] := -1.17915; fTable_Be[202, 2] := 0.163557;
    fTable_Be[203, 0] := 109.770; fTable_Be[203, 1] := -1.27829; fTable_Be[203, 2] := 0.165902;
    fTable_Be[204, 0] := 109.900; fTable_Be[204, 1] := -1.33524; fTable_Be[204, 2] := 0.168057;
    fTable_Be[205, 0] := 110.030; fTable_Be[205, 1] := -1.39580; fTable_Be[205, 2] := 0.168777;
    fTable_Be[206, 0] := 110.160; fTable_Be[206, 1] := -1.45968; fTable_Be[206, 2] := 0.171253;
    fTable_Be[207, 0] := 110.270; fTable_Be[207, 1] := -1.51640; fTable_Be[207, 2] := 0.172992;
    fTable_Be[208, 0] := 110.530; fTable_Be[208, 1] := -1.66366; fTable_Be[208, 2] := 0.176080;
    fTable_Be[209, 0] := 110.660; fTable_Be[209, 1] := -1.74613; fTable_Be[209, 2] := 0.179584;
    fTable_Be[210, 0] := 110.770; fTable_Be[210, 1] := -1.81926; fTable_Be[210, 2] := 0.183052;
    fTable_Be[211, 0] := 110.900; fTable_Be[211, 1] := -1.91441; fTable_Be[211, 2] := 0.183759;
    fTable_Be[212, 0] := 111.030; fTable_Be[212, 1] := -2.01892; fTable_Be[212, 2] := 0.188659;
    fTable_Be[213, 0] := 111.150; fTable_Be[213, 1] := -2.12502; fTable_Be[213, 2] := 0.191441;
    fTable_Be[214, 0] := 111.280; fTable_Be[214, 1] := -2.25725; fTable_Be[214, 2] := 0.192239;
    fTable_Be[215, 0] := 111.400; fTable_Be[215, 1] := -2.40087; fTable_Be[215, 2] := 0.199075;
    fTable_Be[216, 0] := 111.530; fTable_Be[216, 1] := -2.58708; fTable_Be[216, 2] := 0.209517;
    fTable_Be[217, 0] := 111.600; fTable_Be[217, 1] := -2.70637; fTable_Be[217, 2] := 0.223326;
    fTable_Be[218, 0] := 111.800; fTable_Be[218, 1] := -3.21583; fTable_Be[218, 2] := 0.378238;
    fTable_Be[219, 0] := 112.000; fTable_Be[219, 1] := -3.42252; fTable_Be[219, 2] := 1.03860;
    fTable_Be[220, 0] := 112.250; fTable_Be[220, 1] := -3.41684; fTable_Be[220, 2] := 1.38190;
    fTable_Be[221, 0] := 112.500; fTable_Be[221, 1] := -3.59292; fTable_Be[221, 2] := 1.57501;
    fTable_Be[222, 0] := 112.750; fTable_Be[222, 1] := -3.95038; fTable_Be[222, 2] := 2.03965;
    fTable_Be[223, 0] := 113.000; fTable_Be[223, 1] := -3.99197; fTable_Be[223, 2] := 3.05986;
    fTable_Be[224, 0] := 113.250; fTable_Be[224, 1] := -3.32582; fTable_Be[224, 2] := 4.01793;
    fTable_Be[225, 0] := 113.500; fTable_Be[225, 1] := -2.38510; fTable_Be[225, 2] := 4.15418;
    fTable_Be[226, 0] := 113.750; fTable_Be[226, 1] := -1.77257; fTable_Be[226, 2] := 3.84564;
    fTable_Be[227, 0] := 114.000; fTable_Be[227, 1] := -1.49267; fTable_Be[227, 2] := 3.56793;
    fTable_Be[228, 0] := 114.250; fTable_Be[228, 1] := -1.40646; fTable_Be[228, 2] := 3.26353;
    fTable_Be[229, 0] := 114.500; fTable_Be[229, 1] := -1.45558; fTable_Be[229, 2] := 3.11127;
    fTable_Be[230, 0] := 114.750; fTable_Be[230, 1] := -1.51462; fTable_Be[230, 2] := 3.06546;
    fTable_Be[231, 0] := 115.000; fTable_Be[231, 1] := -1.58085; fTable_Be[231, 2] := 3.03372;
    fTable_Be[232, 0] := 115.500; fTable_Be[232, 1] := -1.68141; fTable_Be[232, 2] := 3.14487;
    fTable_Be[233, 0] := 115.750; fTable_Be[233, 1] := -1.68766; fTable_Be[233, 2] := 3.23324;
    fTable_Be[234, 0] := 116.000; fTable_Be[234, 1] := -1.67443; fTable_Be[234, 2] := 3.28469;
    fTable_Be[235, 0] := 116.250; fTable_Be[235, 1] := -1.69668; fTable_Be[235, 2] := 3.30771;
    fTable_Be[236, 0] := 116.500; fTable_Be[236, 1] := -1.74476; fTable_Be[236, 2] := 3.36223;
    fTable_Be[237, 0] := 116.750; fTable_Be[237, 1] := -1.84100; fTable_Be[237, 2] := 3.42546;
    fTable_Be[238, 0] := 117.000; fTable_Be[238, 1] := -1.91971; fTable_Be[238, 2] := 3.58866;
    fTable_Be[239, 0] := 117.250; fTable_Be[239, 1] := -2.01798; fTable_Be[239, 2] := 3.75177;
    fTable_Be[240, 0] := 117.500; fTable_Be[240, 1] := -2.09181; fTable_Be[240, 2] := 4.02099;
    fTable_Be[241, 0] := 117.750; fTable_Be[241, 1] := -1.98599; fTable_Be[241, 2] := 4.48576;
    fTable_Be[242, 0] := 118.000; fTable_Be[242, 1] := -1.69069; fTable_Be[242, 2] := 4.69519;
    fTable_Be[243, 0] := 118.250; fTable_Be[243, 1] := -1.41511; fTable_Be[243, 2] := 4.80543;
    fTable_Be[244, 0] := 118.500; fTable_Be[244, 1] := -1.17170; fTable_Be[244, 2] := 4.79021;
    fTable_Be[245, 0] := 118.750; fTable_Be[245, 1] := -1.03307; fTable_Be[245, 2] := 4.76242;
    fTable_Be[246, 0] := 119.000; fTable_Be[246, 1] := -0.919695; fTable_Be[246, 2] := 4.72326;
    fTable_Be[247, 0] := 119.250; fTable_Be[247, 1] := -0.899806; fTable_Be[247, 2] := 4.70943;
    fTable_Be[248, 0] := 119.500; fTable_Be[248, 1] := -0.833607; fTable_Be[248, 2] := 4.73952;
    fTable_Be[249, 0] := 120.500; fTable_Be[249, 1] := -0.607801; fTable_Be[249, 2] := 5.01171;
    fTable_Be[250, 0] := 121.000; fTable_Be[250, 1] := -0.546931; fTable_Be[250, 2] := 4.97342;
    fTable_Be[251, 0] := 121.500; fTable_Be[251, 1] := -0.418154; fTable_Be[251, 2] := 5.37885;
    fTable_Be[252, 0] := 122.000; fTable_Be[252, 1] := -0.0951663; fTable_Be[252, 2] := 5.50733;
    fTable_Be[253, 0] := 122.500; fTable_Be[253, 1] := 0.195563; fTable_Be[253, 2] := 5.47638;
    fTable_Be[254, 0] := 123.000; fTable_Be[254, 1] := 0.287270; fTable_Be[254, 2] := 5.41101;
    fTable_Be[255, 0] := 123.500; fTable_Be[255, 1] := 0.285511; fTable_Be[255, 2] := 5.46448;
    fTable_Be[256, 0] := 124.000; fTable_Be[256, 1] := 0.326778; fTable_Be[256, 2] := 5.80078;
    fTable_Be[257, 0] := 125.000; fTable_Be[257, 1] := 0.899833; fTable_Be[257, 2] := 6.30269;
    fTable_Be[258, 0] := 125.500; fTable_Be[258, 1] := 1.34102; fTable_Be[258, 2] := 6.64803;
    fTable_Be[259, 0] := 126.000; fTable_Be[259, 1] := 1.95659; fTable_Be[259, 2] := 6.68559;
    fTable_Be[260, 0] := 126.500; fTable_Be[260, 1] := 2.54905; fTable_Be[260, 2] := 6.64790;
    fTable_Be[261, 0] := 127.000; fTable_Be[261, 1] := 3.16414; fTable_Be[261, 2] := 6.40082;
    fTable_Be[262, 0] := 127.500; fTable_Be[262, 1] := 3.67151; fTable_Be[262, 2] := 6.01367;
    fTable_Be[263, 0] := 128.000; fTable_Be[263, 1] := 3.96394; fTable_Be[263, 2] := 5.39328;
    fTable_Be[264, 0] := 128.500; fTable_Be[264, 1] := 4.07172; fTable_Be[264, 2] := 5.00813;
    fTable_Be[265, 0] := 129.000; fTable_Be[265, 1] := 4.14772; fTable_Be[265, 2] := 4.55903;
    fTable_Be[266, 0] := 129.500; fTable_Be[266, 1] := 4.13409; fTable_Be[266, 2] := 4.20865;
    fTable_Be[267, 0] := 130.000; fTable_Be[267, 1] := 4.07072; fTable_Be[267, 2] := 3.82730;
    fTable_Be[268, 0] := 130.500; fTable_Be[268, 1] := 3.96867; fTable_Be[268, 2] := 3.59578;
    fTable_Be[269, 0] := 131.000; fTable_Be[269, 1] := 3.81583; fTable_Be[269, 2] := 3.26529;
    fTable_Be[270, 0] := 131.500; fTable_Be[270, 1] := 3.62226; fTable_Be[270, 2] := 3.15721;
    fTable_Be[271, 0] := 132.000; fTable_Be[271, 1] := 3.45638; fTable_Be[271, 2] := 3.02786;
    fTable_Be[272, 0] := 133.000; fTable_Be[272, 1] := 3.17671; fTable_Be[272, 2] := 2.92660;
    fTable_Be[273, 0] := 133.500; fTable_Be[273, 1] := 3.07605; fTable_Be[273, 2] := 2.93560;
    fTable_Be[274, 0] := 134.000; fTable_Be[274, 1] := 3.00843; fTable_Be[274, 2] := 2.93684;
    fTable_Be[275, 0] := 134.500; fTable_Be[275, 1] := 2.96221; fTable_Be[275, 2] := 2.94578;
    fTable_Be[276, 0] := 135.500; fTable_Be[276, 1] := 2.89396; fTable_Be[276, 2] := 2.93779;
    fTable_Be[277, 0] := 136.000; fTable_Be[277, 1] := 2.87584; fTable_Be[277, 2] := 2.94397;
    fTable_Be[278, 0] := 136.500; fTable_Be[278, 1] := 2.86874; fTable_Be[278, 2] := 2.93959;
    fTable_Be[279, 0] := 137.500; fTable_Be[279, 1] := 2.85627; fTable_Be[279, 2] := 2.89893;
    fTable_Be[280, 0] := 138.000; fTable_Be[280, 1] := 2.83336; fTable_Be[280, 2] := 2.87398;
    fTable_Be[281, 0] := 138.500; fTable_Be[281, 1] := 2.81506; fTable_Be[281, 2] := 2.87098;
    fTable_Be[282, 0] := 139.000; fTable_Be[282, 1] := 2.79734; fTable_Be[282, 2] := 2.84887;
    fTable_Be[283, 0] := 140.000; fTable_Be[283, 1] := 2.73715; fTable_Be[283, 2] := 2.83539;
    fTable_Be[284, 0] := 141.000; fTable_Be[284, 1] := 2.69982; fTable_Be[284, 2] := 2.87711;
    fTable_Be[285, 0] := 141.500; fTable_Be[285, 1] := 2.70638; fTable_Be[285, 2] := 2.90329;
    fTable_Be[286, 0] := 142.000; fTable_Be[286, 1] := 2.71550; fTable_Be[286, 2] := 2.90287;
    fTable_Be[287, 0] := 142.500; fTable_Be[287, 1] := 2.72019; fTable_Be[287, 2] := 2.91465;
    fTable_Be[288, 0] := 143.000; fTable_Be[288, 1] := 2.72987; fTable_Be[288, 2] := 2.91685;
    fTable_Be[289, 0] := 143.500; fTable_Be[289, 1] := 2.74333; fTable_Be[289, 2] := 2.92650;
    fTable_Be[290, 0] := 144.000; fTable_Be[290, 1] := 2.75592; fTable_Be[290, 2] := 2.91495;
    fTable_Be[291, 0] := 144.500; fTable_Be[291, 1] := 2.76383; fTable_Be[291, 2] := 2.91585;
    fTable_Be[292, 0] := 145.000; fTable_Be[292, 1] := 2.76841; fTable_Be[292, 2] := 2.90262;
    fTable_Be[293, 0] := 145.500; fTable_Be[293, 1] := 2.77007; fTable_Be[293, 2] := 2.90346;
    fTable_Be[294, 0] := 146.000; fTable_Be[294, 1] := 2.76964; fTable_Be[294, 2] := 2.89577;
    fTable_Be[295, 0] := 146.500; fTable_Be[295, 1] := 2.76561; fTable_Be[295, 2] := 2.89537;
    fTable_Be[296, 0] := 148.000; fTable_Be[296, 1] := 2.76343; fTable_Be[296, 2] := 2.93154;
    fTable_Be[297, 0] := 148.500; fTable_Be[297, 1] := 2.77483; fTable_Be[297, 2] := 2.94822;
    fTable_Be[298, 0] := 149.000; fTable_Be[298, 1] := 2.78740; fTable_Be[298, 2] := 2.95243;
    fTable_Be[299, 0] := 150.000; fTable_Be[299, 1] := 2.81919; fTable_Be[299, 2] := 2.98597;
    fTable_Be[300, 0] := 151.000; fTable_Be[300, 1] := 2.85322; fTable_Be[300, 2] := 2.98029;
    fTable_Be[301, 0] := 152.000; fTable_Be[301, 1] := 2.86818; fTable_Be[301, 2] := 2.98203;
    fTable_Be[302, 0] := 153.000; fTable_Be[302, 1] := 2.89266; fTable_Be[302, 2] := 3.01367;
    fTable_Be[303, 0] := 153.500; fTable_Be[303, 1] := 2.89847; fTable_Be[303, 2] := 3.01671;
    fTable_Be[304, 0] := 155.000; fTable_Be[304, 1] := 2.93623; fTable_Be[304, 2] := 3.06074;
    fTable_Be[305, 0] := 155.500; fTable_Be[305, 1] := 2.96092; fTable_Be[305, 2] := 3.08803;
    fTable_Be[306, 0] := 156.500; fTable_Be[306, 1] := 3.01251; fTable_Be[306, 2] := 3.12840;
    fTable_Be[307, 0] := 157.000; fTable_Be[307, 1] := 3.04430; fTable_Be[307, 2] := 3.14926;
    fTable_Be[308, 0] := 157.500; fTable_Be[308, 1] := 3.08675; fTable_Be[308, 2] := 3.17679;
    fTable_Be[309, 0] := 158.000; fTable_Be[309, 1] := 3.13492; fTable_Be[309, 2] := 3.18715;
    fTable_Be[310, 0] := 159.000; fTable_Be[310, 1] := 3.22830; fTable_Be[310, 2] := 3.19053;
    fTable_Be[311, 0] := 160.000; fTable_Be[311, 1] := 3.32359; fTable_Be[311, 2] := 3.19716;
    fTable_Be[312, 0] := 160.500; fTable_Be[312, 1] := 3.37652; fTable_Be[312, 2] := 3.19224;
    fTable_Be[313, 0] := 161.500; fTable_Be[313, 1] := 3.48313; fTable_Be[313, 2] := 3.16079;
    fTable_Be[314, 0] := 162.000; fTable_Be[314, 1] := 3.53440; fTable_Be[314, 2] := 3.15119;
    fTable_Be[315, 0] := 163.000; fTable_Be[315, 1] := 3.64004; fTable_Be[315, 2] := 3.07868;
    fTable_Be[316, 0] := 164.500; fTable_Be[316, 1] := 3.74596; fTable_Be[316, 2] := 2.93822;
    fTable_Be[317, 0] := 165.500; fTable_Be[317, 1] := 3.78278; fTable_Be[317, 2] := 2.85215;
    fTable_Be[318, 0] := 166.000; fTable_Be[318, 1] := 3.79484; fTable_Be[318, 2] := 2.81725;
    fTable_Be[319, 0] := 167.000; fTable_Be[319, 1] := 3.82135; fTable_Be[319, 2] := 2.73264;
    fTable_Be[320, 0] := 167.500; fTable_Be[320, 1] := 3.82362; fTable_Be[320, 2] := 2.69680;
    fTable_Be[321, 0] := 168.000; fTable_Be[321, 1] := 3.81959; fTable_Be[321, 2] := 2.65488;
    fTable_Be[322, 0] := 169.500; fTable_Be[322, 1] := 3.80124; fTable_Be[322, 2] := 2.57094;
    fTable_Be[323, 0] := 170.000; fTable_Be[323, 1] := 3.79268; fTable_Be[323, 2] := 2.55180;
    fTable_Be[324, 0] := 170.500; fTable_Be[324, 1] := 3.78838; fTable_Be[324, 2] := 2.54214;
    fTable_Be[325, 0] := 171.000; fTable_Be[325, 1] := 3.78748; fTable_Be[325, 2] := 2.52605;
    fTable_Be[326, 0] := 171.500; fTable_Be[326, 1] := 3.78804; fTable_Be[326, 2] := 2.51896;
    fTable_Be[327, 0] := 172.990; fTable_Be[327, 1] := 3.80814; fTable_Be[327, 2] := 2.47360;
    fTable_Be[328, 0] := 173.990; fTable_Be[328, 1] := 3.80347; fTable_Be[328, 2] := 2.43390;
    fTable_Be[329, 0] := 174.500; fTable_Be[329, 1] := 3.81339; fTable_Be[329, 2] := 2.43394;
    fTable_Be[330, 0] := 175.510; fTable_Be[330, 1] := 3.82900; fTable_Be[330, 2] := 2.40213;
    fTable_Be[331, 0] := 176.000; fTable_Be[331, 1] := 3.83339; fTable_Be[331, 2] := 2.38083;
    fTable_Be[332, 0] := 176.500; fTable_Be[332, 1] := 3.83871; fTable_Be[332, 2] := 2.36562;
    fTable_Be[333, 0] := 177.510; fTable_Be[333, 1] := 3.85216; fTable_Be[333, 2] := 2.32073;
    fTable_Be[334, 0] := 178.000; fTable_Be[334, 1] := 3.84430; fTable_Be[334, 2] := 2.28306;
    fTable_Be[335, 0] := 178.500; fTable_Be[335, 1] := 3.84361; fTable_Be[335, 2] := 2.27434;
    fTable_Be[336, 0] := 180.000; fTable_Be[336, 1] := 3.79942; fTable_Be[336, 2] := 2.22984;
    fTable_Be[337, 0] := 181.000; fTable_Be[337, 1] := 3.78489; fTable_Be[337, 2] := 2.22505;
    fTable_Be[338, 0] := 181.510; fTable_Be[338, 1] := 3.78464; fTable_Be[338, 2] := 2.22872;
    fTable_Be[339, 0] := 182.000; fTable_Be[339, 1] := 3.77923; fTable_Be[339, 2] := 2.21064;
    fTable_Be[340, 0] := 183.500; fTable_Be[340, 1] := 3.77455; fTable_Be[340, 2] := 2.19974;
    fTable_Be[341, 0] := 184.490; fTable_Be[341, 1] := 3.77588; fTable_Be[341, 2] := 2.18992;
    fTable_Be[342, 0] := 187.474; fTable_Be[342, 1] := 3.78737; fTable_Be[342, 2] := 2.16785;
    fTable_Be[343, 0] := 187.500; fTable_Be[343, 1] := 3.78737; fTable_Be[343, 2] := 2.16766;
    fTable_Be[344, 0] := 188.000; fTable_Be[344, 1] := 3.77910; fTable_Be[344, 2] := 2.15580;
    fTable_Be[345, 0] := 188.500; fTable_Be[345, 1] := 3.77675; fTable_Be[345, 2] := 2.16037;
    fTable_Be[346, 0] := 189.000; fTable_Be[346, 1] := 3.77711; fTable_Be[346, 2] := 2.15869;
    fTable_Be[347, 0] := 190.000; fTable_Be[347, 1] := 3.78555; fTable_Be[347, 2] := 2.16413;
    fTable_Be[348, 0] := 190.500; fTable_Be[348, 1] := 3.79166; fTable_Be[348, 2] := 2.15995;
    fTable_Be[349, 0] := 191.000; fTable_Be[349, 1] := 3.79603; fTable_Be[349, 2] := 2.16059;
    fTable_Be[350, 0] := 192.000; fTable_Be[350, 1] := 3.80715; fTable_Be[350, 2] := 2.14936;
    fTable_Be[351, 0] := 193.510; fTable_Be[351, 1] := 3.82898; fTable_Be[351, 2] := 2.14231;
    fTable_Be[352, 0] := 194.000; fTable_Be[352, 1] := 3.83942; fTable_Be[352, 2] := 2.13531;
    fTable_Be[353, 0] := 194.500; fTable_Be[353, 1] := 3.84007; fTable_Be[353, 2] := 2.11653;
    fTable_Be[354, 0] := 195.000; fTable_Be[354, 1] := 3.83469; fTable_Be[354, 2] := 2.11378;
    fTable_Be[355, 0] := 195.500; fTable_Be[355, 1] := 3.83653; fTable_Be[355, 2] := 2.11602;
    fTable_Be[356, 0] := 196.500; fTable_Be[356, 1] := 3.84812; fTable_Be[356, 2] := 2.10677;
    fTable_Be[357, 0] := 197.500; fTable_Be[357, 1] := 3.85281; fTable_Be[357, 2] := 2.09245;
    fTable_Be[358, 0] := 199.010; fTable_Be[358, 1] := 3.86036; fTable_Be[358, 2] := 2.09404;
    fTable_Be[359, 0] := 200.000; fTable_Be[359, 1] := 3.87172; fTable_Be[359, 2] := 2.08193;
    fTable_Be[360, 0] := 201.500; fTable_Be[360, 1] := 3.88191; fTable_Be[360, 2] := 2.07385;
    fTable_Be[361, 0] := 203.000; fTable_Be[361, 1] := 3.89450; fTable_Be[361, 2] := 2.07146;
    fTable_Be[362, 0] := 204.500; fTable_Be[362, 1] := 3.92105; fTable_Be[362, 2] := 2.06855;
    fTable_Be[363, 0] := 207.000; fTable_Be[363, 1] := 3.96780; fTable_Be[363, 2] := 2.04405;
    fTable_Be[364, 0] := 207.500; fTable_Be[364, 1] := 3.97172; fTable_Be[364, 2] := 2.03179;
    fTable_Be[365, 0] := 208.010; fTable_Be[365, 1] := 3.97628; fTable_Be[365, 2] := 2.03019;
    fTable_Be[366, 0] := 208.500; fTable_Be[366, 1] := 3.97935; fTable_Be[366, 2] := 2.02063;
    fTable_Be[367, 0] := 210.500; fTable_Be[367, 1] := 4.00635; fTable_Be[367, 2] := 2.00156;
    fTable_Be[368, 0] := 212.000; fTable_Be[368, 1] := 4.02425; fTable_Be[368, 2] := 1.97791;
    fTable_Be[369, 0] := 212.500; fTable_Be[369, 1] := 4.02760; fTable_Be[369, 2] := 1.97716;
    fTable_Be[370, 0] := 213.000; fTable_Be[370, 1] := 4.03863; fTable_Be[370, 2] := 1.96995;
    fTable_Be[371, 0] := 213.500; fTable_Be[371, 1] := 4.04264; fTable_Be[371, 2] := 1.95601;
    fTable_Be[372, 0] := 214.500; fTable_Be[372, 1] := 4.04244; fTable_Be[372, 2] := 1.94417;
    fTable_Be[373, 0] := 215.000; fTable_Be[373, 1] := 4.04818; fTable_Be[373, 2] := 1.94719;
    fTable_Be[374, 0] := 215.500; fTable_Be[374, 1] := 4.05146; fTable_Be[374, 2] := 1.93625;
    fTable_Be[375, 0] := 217.000; fTable_Be[375, 1] := 4.07177; fTable_Be[375, 2] := 1.91827;
    fTable_Be[376, 0] := 218.000; fTable_Be[376, 1] := 4.07937; fTable_Be[376, 2] := 1.90175;
    fTable_Be[377, 0] := 219.000; fTable_Be[377, 1] := 4.08572; fTable_Be[377, 2] := 1.89162;
    fTable_Be[378, 0] := 220.000; fTable_Be[378, 1] := 4.09161; fTable_Be[378, 2] := 1.87778;
    fTable_Be[379, 0] := 220.500; fTable_Be[379, 1] := 4.09066; fTable_Be[379, 2] := 1.87308;
    fTable_Be[380, 0] := 221.000; fTable_Be[380, 1] := 4.09659; fTable_Be[380, 2] := 1.87799;
    fTable_Be[381, 0] := 221.500; fTable_Be[381, 1] := 4.10445; fTable_Be[381, 2] := 1.86891;
    fTable_Be[382, 0] := 222.000; fTable_Be[382, 1] := 4.11052; fTable_Be[382, 2] := 1.86480;
    fTable_Be[383, 0] := 222.500; fTable_Be[383, 1] := 4.11500; fTable_Be[383, 2] := 1.85638;
    fTable_Be[384, 0] := 223.000; fTable_Be[384, 1] := 4.12075; fTable_Be[384, 2] := 1.85152;
    fTable_Be[385, 0] := 223.500; fTable_Be[385, 1] := 4.12176; fTable_Be[385, 2] := 1.84131;
    fTable_Be[386, 0] := 224.000; fTable_Be[386, 1] := 4.12134; fTable_Be[386, 2] := 1.83756;
    fTable_Be[387, 0] := 224.500; fTable_Be[387, 1] := 4.12348; fTable_Be[387, 2] := 1.84253;
    fTable_Be[388, 0] := 226.000; fTable_Be[388, 1] := 4.15704; fTable_Be[388, 2] := 1.82599;
    fTable_Be[389, 0] := 226.490; fTable_Be[389, 1] := 4.16101; fTable_Be[389, 2] := 1.81782;
    fTable_Be[390, 0] := 227.500; fTable_Be[390, 1] := 4.17850; fTable_Be[390, 2] := 1.80946;
    fTable_Be[391, 0] := 228.000; fTable_Be[391, 1] := 4.19190; fTable_Be[391, 2] := 1.79537;
    fTable_Be[392, 0] := 228.500; fTable_Be[392, 1] := 4.19439; fTable_Be[392, 2] := 1.77053;
    fTable_Be[393, 0] := 229.000; fTable_Be[393, 1] := 4.19072; fTable_Be[393, 2] := 1.76739;
    fTable_Be[394, 0] := 229.500; fTable_Be[394, 1] := 4.19374; fTable_Be[394, 2] := 1.75778;
    fTable_Be[395, 0] := 230.500; fTable_Be[395, 1] := 4.19691; fTable_Be[395, 2] := 1.74263;
    fTable_Be[396, 0] := 231.000; fTable_Be[396, 1] := 4.20734; fTable_Be[396, 2] := 1.73860;
    fTable_Be[397, 0] := 231.500; fTable_Be[397, 1] := 4.21071; fTable_Be[397, 2] := 1.72476;
    fTable_Be[398, 0] := 232.000; fTable_Be[398, 1] := 4.21210; fTable_Be[398, 2] := 1.70717;
    fTable_Be[399, 0] := 234.500; fTable_Be[399, 1] := 4.21500; fTable_Be[399, 2] := 1.66650;
    fTable_Be[400, 0] := 235.000; fTable_Be[400, 1] := 4.20480; fTable_Be[400, 2] := 1.65173;
    fTable_Be[401, 0] := 235.500; fTable_Be[401, 1] := 4.20096; fTable_Be[401, 2] := 1.64949;
    fTable_Be[402, 0] := 236.500; fTable_Be[402, 1] := 4.20132; fTable_Be[402, 2] := 1.65027;
    fTable_Be[403, 0] := 237.500; fTable_Be[403, 1] := 4.20371; fTable_Be[403, 2] := 1.63115;
    fTable_Be[404, 0] := 238.000; fTable_Be[404, 1] := 4.20288; fTable_Be[404, 2] := 1.62857;
    fTable_Be[405, 0] := 238.500; fTable_Be[405, 1] := 4.20322; fTable_Be[405, 2] := 1.62029;
    fTable_Be[406, 0] := 239.500; fTable_Be[406, 1] := 4.20097; fTable_Be[406, 2] := 1.61693;
    fTable_Be[407, 0] := 240.000; fTable_Be[407, 1] := 4.20624; fTable_Be[407, 2] := 1.61172;
    fTable_Be[408, 0] := 240.500; fTable_Be[408, 1] := 4.20812; fTable_Be[408, 2] := 1.60246;
    fTable_Be[409, 0] := 241.000; fTable_Be[409, 1] := 4.21110; fTable_Be[409, 2] := 1.59846;
    fTable_Be[410, 0] := 241.500; fTable_Be[410, 1] := 4.20782; fTable_Be[410, 2] := 1.58125;
    fTable_Be[411, 0] := 242.000; fTable_Be[411, 1] := 4.19755; fTable_Be[411, 2] := 1.57866;
    fTable_Be[412, 0] := 242.500; fTable_Be[412, 1] := 4.19930; fTable_Be[412, 2] := 1.58572;
    fTable_Be[413, 0] := 243.500; fTable_Be[413, 1] := 4.21118; fTable_Be[413, 2] := 1.57948;
    fTable_Be[414, 0] := 244.000; fTable_Be[414, 1] := 4.20763; fTable_Be[414, 2] := 1.56140;
    fTable_Be[415, 0] := 244.500; fTable_Be[415, 1] := 4.20246; fTable_Be[415, 2] := 1.56099;
    fTable_Be[416, 0] := 245.000; fTable_Be[416, 1] := 4.19678; fTable_Be[416, 2] := 1.55568;
    fTable_Be[417, 0] := 246.000; fTable_Be[417, 1] := 4.19512; fTable_Be[417, 2] := 1.55713;
    fTable_Be[418, 0] := 246.500; fTable_Be[418, 1] := 4.19511; fTable_Be[418, 2] := 1.55644;
    fTable_Be[419, 0] := 247.500; fTable_Be[419, 1] := 4.19613; fTable_Be[419, 2] := 1.55114;
    fTable_Be[420, 0] := 248.500; fTable_Be[420, 1] := 4.18859; fTable_Be[420, 2] := 1.55086;
    fTable_Be[421, 0] := 248.990; fTable_Be[421, 1] := 4.19626; fTable_Be[421, 2] := 1.56821;
    fTable_Be[422, 0] := 249.500; fTable_Be[422, 1] := 4.21213; fTable_Be[422, 2] := 1.56785;
    fTable_Be[423, 0] := 250.000; fTable_Be[423, 1] := 4.22653; fTable_Be[423, 2] := 1.55043;
    fTable_Be[424, 0] := 251.540; fTable_Be[424, 1] := 4.26661; fTable_Be[424, 2] := 1.54085;
    fTable_Be[425, 0] := 255.608; fTable_Be[425, 1] := 4.25156; fTable_Be[425, 2] := 1.50042;
    fTable_Be[426, 0] := 259.743; fTable_Be[426, 1] := 4.26764; fTable_Be[426, 2] := 1.46106;
    fTable_Be[427, 0] := 263.944; fTable_Be[427, 1] := 4.28045; fTable_Be[427, 2] := 1.42272;
    fTable_Be[428, 0] := 268.213; fTable_Be[428, 1] := 4.29117; fTable_Be[428, 2] := 1.38539;
    fTable_Be[429, 0] := 272.551; fTable_Be[429, 1] := 4.30032; fTable_Be[429, 2] := 1.34904;
    fTable_Be[430, 0] := 276.959; fTable_Be[430, 1] := 4.30821; fTable_Be[430, 2] := 1.31364;
    fTable_Be[431, 0] := 281.439; fTable_Be[431, 1] := 4.31501; fTable_Be[431, 2] := 1.27917;
    fTable_Be[432, 0] := 285.991; fTable_Be[432, 1] := 4.32087; fTable_Be[432, 2] := 1.24561;
    fTable_Be[433, 0] := 290.617; fTable_Be[433, 1] := 4.32588; fTable_Be[433, 2] := 1.21293;
    fTable_Be[434, 0] := 295.317; fTable_Be[434, 1] := 4.33013; fTable_Be[434, 2] := 1.18110;
    fTable_Be[435, 0] := 300.094; fTable_Be[435, 1] := 4.33368; fTable_Be[435, 2] := 1.15011;
    fTable_Be[436, 0] := 304.947; fTable_Be[436, 1] := 4.33653; fTable_Be[436, 2] := 1.11993;
    fTable_Be[437, 0] := 309.880; fTable_Be[437, 1] := 4.33874; fTable_Be[437, 2] := 1.09055;
    fTable_Be[438, 0] := 314.892; fTable_Be[438, 1] := 4.34029; fTable_Be[438, 2] := 1.06193;
    fTable_Be[439, 0] := 319.985; fTable_Be[439, 1] := 4.34126; fTable_Be[439, 2] := 1.03488;
    fTable_Be[440, 0] := 325.160; fTable_Be[440, 1] := 4.34227; fTable_Be[440, 2] := 1.00851;
    fTable_Be[441, 0] := 330.420; fTable_Be[441, 1] := 4.34307; fTable_Be[441, 2] := 0.982821;
    fTable_Be[442, 0] := 335.764; fTable_Be[442, 1] := 4.34364; fTable_Be[442, 2] := 0.957781;
    fTable_Be[443, 0] := 341.195; fTable_Be[443, 1] := 4.34399; fTable_Be[443, 2] := 0.933380;
    fTable_Be[444, 0] := 346.713; fTable_Be[444, 1] := 4.34413; fTable_Be[444, 2] := 0.909600;
    fTable_Be[445, 0] := 352.321; fTable_Be[445, 1] := 4.34408; fTable_Be[445, 2] := 0.886427;
    fTable_Be[446, 0] := 358.020; fTable_Be[446, 1] := 4.34387; fTable_Be[446, 2] := 0.863843;
    fTable_Be[447, 0] := 363.810; fTable_Be[447, 1] := 4.34352; fTable_Be[447, 2] := 0.841835;
    fTable_Be[448, 0] := 369.695; fTable_Be[448, 1] := 4.34307; fTable_Be[448, 2] := 0.820388;
    fTable_Be[449, 0] := 375.674; fTable_Be[449, 1] := 4.34247; fTable_Be[449, 2] := 0.799486;
    fTable_Be[450, 0] := 381.750; fTable_Be[450, 1] := 4.34234; fTable_Be[450, 2] := 0.779118;
    fTable_Be[451, 0] := 387.925; fTable_Be[451, 1] := 4.34238; fTable_Be[451, 2] := 0.759267;
    fTable_Be[452, 0] := 394.199; fTable_Be[452, 1] := 4.34228; fTable_Be[452, 2] := 0.738576;
    fTable_Be[453, 0] := 400.575; fTable_Be[453, 1] := 4.34177; fTable_Be[453, 2] := 0.718448;
    fTable_Be[454, 0] := 407.054; fTable_Be[454, 1] := 4.34059; fTable_Be[454, 2] := 0.697922;
    fTable_Be[455, 0] := 413.638; fTable_Be[455, 1] := 4.33897; fTable_Be[455, 2] := 0.677984;
    fTable_Be[456, 0] := 420.328; fTable_Be[456, 1] := 4.33688; fTable_Be[456, 2] := 0.658616;
    fTable_Be[457, 0] := 427.126; fTable_Be[457, 1] := 4.33438; fTable_Be[457, 2] := 0.639799;
    fTable_Be[458, 0] := 434.035; fTable_Be[458, 1] := 4.33165; fTable_Be[458, 2] := 0.621521;
    fTable_Be[459, 0] := 441.055; fTable_Be[459, 1] := 4.32870; fTable_Be[459, 2] := 0.603766;
    fTable_Be[460, 0] := 448.189; fTable_Be[460, 1] := 4.32557; fTable_Be[460, 2] := 0.586516;
    fTable_Be[461, 0] := 455.438; fTable_Be[461, 1] := 4.32228; fTable_Be[461, 2] := 0.569761;
    fTable_Be[462, 0] := 462.804; fTable_Be[462, 1] := 4.31886; fTable_Be[462, 2] := 0.553484;
    fTable_Be[463, 0] := 470.290; fTable_Be[463, 1] := 4.31532; fTable_Be[463, 2] := 0.537671;
    fTable_Be[464, 0] := 477.896; fTable_Be[464, 1] := 4.31169; fTable_Be[464, 2] := 0.522311;
    fTable_Be[465, 0] := 485.626; fTable_Be[465, 1] := 4.30798; fTable_Be[465, 2] := 0.507390;
    fTable_Be[466, 0] := 493.480; fTable_Be[466, 1] := 4.30421; fTable_Be[466, 2] := 0.492894;
    fTable_Be[467, 0] := 501.462; fTable_Be[467, 1] := 4.30038; fTable_Be[467, 2] := 0.478813;
    fTable_Be[468, 0] := 509.573; fTable_Be[468, 1] := 4.29651; fTable_Be[468, 2] := 0.465133;
    fTable_Be[469, 0] := 517.815; fTable_Be[469, 1] := 4.29262; fTable_Be[469, 2] := 0.451845;
    fTable_Be[470, 0] := 526.190; fTable_Be[470, 1] := 4.28871; fTable_Be[470, 2] := 0.438937;
    fTable_Be[471, 0] := 534.701; fTable_Be[471, 1] := 4.28480; fTable_Be[471, 2] := 0.426397;
    fTable_Be[472, 0] := 543.349; fTable_Be[472, 1] := 4.28091; fTable_Be[472, 2] := 0.414215;
    fTable_Be[473, 0] := 552.137; fTable_Be[473, 1] := 4.27707; fTable_Be[473, 2] := 0.402382;
    fTable_Be[474, 0] := 561.068; fTable_Be[474, 1] := 4.27342; fTable_Be[474, 2] := 0.390887;
    fTable_Be[475, 0] := 570.142; fTable_Be[475, 1] := 4.26964; fTable_Be[475, 2] := 0.379297;
    fTable_Be[476, 0] := 579.364; fTable_Be[476, 1] := 4.26575; fTable_Be[476, 2] := 0.368051;
    fTable_Be[477, 0] := 588.735; fTable_Be[477, 1] := 4.26181; fTable_Be[477, 2] := 0.357139;
    fTable_Be[478, 0] := 598.257; fTable_Be[478, 1] := 4.25782; fTable_Be[478, 2] := 0.346550;
    fTable_Be[479, 0] := 607.933; fTable_Be[479, 1] := 4.25382; fTable_Be[479, 2] := 0.336275;
    fTable_Be[480, 0] := 617.766; fTable_Be[480, 1] := 4.24986; fTable_Be[480, 2] := 0.326305;
    fTable_Be[481, 0] := 627.758; fTable_Be[481, 1] := 4.24601; fTable_Be[481, 2] := 0.316630;
    fTable_Be[482, 0] := 637.912; fTable_Be[482, 1] := 4.24229; fTable_Be[482, 2] := 0.307242;
    fTable_Be[483, 0] := 648.229; fTable_Be[483, 1] := 4.23849; fTable_Be[483, 2] := 0.297321;
    fTable_Be[484, 0] := 658.714; fTable_Be[484, 1] := 4.23444; fTable_Be[484, 2] := 0.287720;
    fTable_Be[485, 0] := 669.368; fTable_Be[485, 1] := 4.22972; fTable_Be[485, 2] := 0.278430;
    fTable_Be[486, 0] := 680.195; fTable_Be[486, 1] := 4.22459; fTable_Be[486, 2] := 0.270148;
    fTable_Be[487, 0] := 691.196; fTable_Be[487, 1] := 4.22029; fTable_Be[487, 2] := 0.262802;
    fTable_Be[488, 0] := 702.376; fTable_Be[488, 1] := 4.21661; fTable_Be[488, 2] := 0.255654;
    fTable_Be[489, 0] := 713.736; fTable_Be[489, 1] := 4.21310; fTable_Be[489, 2] := 0.247975;
    fTable_Be[490, 0] := 725.280; fTable_Be[490, 1] := 4.20947; fTable_Be[490, 2] := 0.240525;
    fTable_Be[491, 0] := 737.011; fTable_Be[491, 1] := 4.20574; fTable_Be[491, 2] := 0.233102;
    fTable_Be[492, 0] := 748.932; fTable_Be[492, 1] := 4.20199; fTable_Be[492, 2] := 0.225907;
    fTable_Be[493, 0] := 761.045; fTable_Be[493, 1] := 4.19823; fTable_Be[493, 2] := 0.218934;
    fTable_Be[494, 0] := 773.354; fTable_Be[494, 1] := 4.19446; fTable_Be[494, 2] := 0.212177;
    fTable_Be[495, 0] := 785.863; fTable_Be[495, 1] := 4.19072; fTable_Be[495, 2] := 0.205628;
    fTable_Be[496, 0] := 798.573; fTable_Be[496, 1] := 4.18700; fTable_Be[496, 2] := 0.199281;
    fTable_Be[497, 0] := 811.490; fTable_Be[497, 1] := 4.18331; fTable_Be[497, 2] := 0.193131;
    fTable_Be[498, 0] := 824.615; fTable_Be[498, 1] := 4.17967; fTable_Be[498, 2] := 0.187170;
    fTable_Be[499, 0] := 837.952; fTable_Be[499, 1] := 4.17606; fTable_Be[499, 2] := 0.181392;
    fTable_Be[500, 0] := 851.505; fTable_Be[500, 1] := 4.17249; fTable_Be[500, 2] := 0.175794;
    fTable_Be[501, 0] := 865.278; fTable_Be[501, 1] := 4.16897; fTable_Be[501, 2] := 0.170368;
    fTable_Be[502, 0] := 879.273; fTable_Be[502, 1] := 4.16547; fTable_Be[502, 2] := 0.165110;
    fTable_Be[503, 0] := 893.495; fTable_Be[503, 1] := 4.16203; fTable_Be[503, 2] := 0.160057;
    fTable_Be[504, 0] := 907.946; fTable_Be[504, 1] := 4.15866; fTable_Be[504, 2] := 0.155160;
    fTable_Be[505, 0] := 922.631; fTable_Be[505, 1] := 4.15540; fTable_Be[505, 2] := 0.150411;
    fTable_Be[506, 0] := 937.554; fTable_Be[506, 1] := 4.15220; fTable_Be[506, 2] := 0.145809;
    fTable_Be[507, 0] := 952.719; fTable_Be[507, 1] := 4.14905; fTable_Be[507, 2] := 0.141250;
    fTable_Be[508, 0] := 968.128; fTable_Be[508, 1] := 4.14591; fTable_Be[508, 2] := 0.136834;
    fTable_Be[509, 0] := 983.787; fTable_Be[509, 1] := 4.14280; fTable_Be[509, 2] := 0.132557;
    fTable_Be[510, 0] := 999.699; fTable_Be[510, 1] := 4.13974; fTable_Be[510, 2] := 0.128412;
    fTable_Be[511, 0] := 1015.87; fTable_Be[511, 1] := 4.13672; fTable_Be[511, 2] := 0.124398;
    fTable_Be[512, 0] := 1032.30; fTable_Be[512, 1] := 4.13375; fTable_Be[512, 2] := 0.120509;
    fTable_Be[513, 0] := 1049; fTable_Be[513, 1] := 4.13082; fTable_Be[513, 2] := 0.116741;
    fTable_Be[514, 0] := 1065.96; fTable_Be[514, 1] := 4.12794; fTable_Be[514, 2] := 0.113091;
    fTable_Be[515, 0] := 1083.20; fTable_Be[515, 1] := 4.12511; fTable_Be[515, 2] := 0.109556;
    fTable_Be[516, 0] := 1100.72; fTable_Be[516, 1] := 4.12233; fTable_Be[516, 2] := 0.106131;
    fTable_Be[517, 0] := 1118.53; fTable_Be[517, 1] := 4.11960; fTable_Be[517, 2] := 0.102813;
    fTable_Be[518, 0] := 1136.62; fTable_Be[518, 1] := 4.11692; fTable_Be[518, 2] := 0.0995984;
    fTable_Be[519, 0] := 1155; fTable_Be[519, 1] := 4.11429; fTable_Be[519, 2] := 0.0964847;
    fTable_Be[520, 0] := 1173.68; fTable_Be[520, 1] := 4.11170; fTable_Be[520, 2] := 0.0934681;
    fTable_Be[521, 0] := 1192.67; fTable_Be[521, 1] := 4.10917; fTable_Be[521, 2] := 0.0905461;
    fTable_Be[522, 0] := 1211.96; fTable_Be[522, 1] := 4.10668; fTable_Be[522, 2] := 0.0877153;
    fTable_Be[523, 0] := 1231.56; fTable_Be[523, 1] := 4.10424; fTable_Be[523, 2] := 0.0849730;
    fTable_Be[524, 0] := 1251.48; fTable_Be[524, 1] := 4.10185; fTable_Be[524, 2] := 0.0823165;
    fTable_Be[525, 0] := 1271.72; fTable_Be[525, 1] := 4.09951; fTable_Be[525, 2] := 0.0797430;
    fTable_Be[526, 0] := 1292.29; fTable_Be[526, 1] := 4.09722; fTable_Be[526, 2] := 0.0772499;
    fTable_Be[527, 0] := 1313.19; fTable_Be[527, 1] := 4.09497; fTable_Be[527, 2] := 0.0748349;
    fTable_Be[528, 0] := 1334.43; fTable_Be[528, 1] := 4.09277; fTable_Be[528, 2] := 0.0724952;
    fTable_Be[529, 0] := 1356.01; fTable_Be[529, 1] := 4.09061; fTable_Be[529, 2] := 0.0702288;
    fTable_Be[530, 0] := 1377.95; fTable_Be[530, 1] := 4.08851; fTable_Be[530, 2] := 0.0680301;
    fTable_Be[531, 0] := 1400.23; fTable_Be[531, 1] := 4.08644; fTable_Be[531, 2] := 0.0659001;
    fTable_Be[532, 0] := 1422.88; fTable_Be[532, 1] := 4.08442; fTable_Be[532, 2] := 0.0638369;
    fTable_Be[533, 0] := 1445.90; fTable_Be[533, 1] := 4.08245; fTable_Be[533, 2] := 0.0618382;
    fTable_Be[534, 0] := 1469.28; fTable_Be[534, 1] := 4.08052; fTable_Be[534, 2] := 0.0599022;
    fTable_Be[535, 0] := 1493.05; fTable_Be[535, 1] := 4.07864; fTable_Be[535, 2] := 0.0580268;
    fTable_Be[536, 0] := 1517.20; fTable_Be[536, 1] := 4.07683; fTable_Be[536, 2] := 0.0562100;
    fTable_Be[537, 0] := 1541.73; fTable_Be[537, 1] := 4.07504; fTable_Be[537, 2] := 0.0543948;
    fTable_Be[538, 0] := 1566.67; fTable_Be[538, 1] := 4.07327; fTable_Be[538, 2] := 0.0526382;
    fTable_Be[539, 0] := 1592.01; fTable_Be[539, 1] := 4.07153; fTable_Be[539, 2] := 0.0509382;
    fTable_Be[540, 0] := 1617.76; fTable_Be[540, 1] := 4.06982; fTable_Be[540, 2] := 0.0492933;
    fTable_Be[541, 0] := 1643.93; fTable_Be[541, 1] := 4.06814; fTable_Be[541, 2] := 0.0477014;
    fTable_Be[542, 0] := 1670.52; fTable_Be[542, 1] := 4.06650; fTable_Be[542, 2] := 0.0461609;
    fTable_Be[543, 0] := 1697.53; fTable_Be[543, 1] := 4.06489; fTable_Be[543, 2] := 0.0446702;
    fTable_Be[544, 0] := 1724.99; fTable_Be[544, 1] := 4.06331; fTable_Be[544, 2] := 0.0432276;
    fTable_Be[545, 0] := 1752.89; fTable_Be[545, 1] := 4.06176; fTable_Be[545, 2] := 0.0418316;
    fTable_Be[546, 0] := 1781.24; fTable_Be[546, 1] := 4.06025; fTable_Be[546, 2] := 0.0404807;
    fTable_Be[547, 0] := 1810.05; fTable_Be[547, 1] := 4.05877; fTable_Be[547, 2] := 0.0391734;
    fTable_Be[548, 0] := 1839.33; fTable_Be[548, 1] := 4.05733; fTable_Be[548, 2] := 0.0379083;
    fTable_Be[549, 0] := 1869.08; fTable_Be[549, 1] := 4.05592; fTable_Be[549, 2] := 0.0366841;
    fTable_Be[550, 0] := 1899.31; fTable_Be[550, 1] := 4.05453; fTable_Be[550, 2] := 0.0354994;
    fTable_Be[551, 0] := 1930.03; fTable_Be[551, 1] := 4.05319; fTable_Be[551, 2] := 0.0343530;
    fTable_Be[552, 0] := 1961.25; fTable_Be[552, 1] := 4.05187; fTable_Be[552, 2] := 0.0332436;
    fTable_Be[553, 0] := 1992.97; fTable_Be[553, 1] := 4.05059; fTable_Be[553, 2] := 0.0321700;
    fTable_Be[554, 0] := 2025.20; fTable_Be[554, 1] := 4.04935; fTable_Be[554, 2] := 0.0311311;
    fTable_Be[555, 0] := 2057.96; fTable_Be[555, 1] := 4.04813; fTable_Be[555, 2] := 0.0300957;
    fTable_Be[556, 0] := 2091.24; fTable_Be[556, 1] := 4.04693; fTable_Be[556, 2] := 0.0290947;
    fTable_Be[557, 0] := 2125.07; fTable_Be[557, 1] := 4.04575; fTable_Be[557, 2] := 0.0281270;
    fTable_Be[558, 0] := 2159.44; fTable_Be[558, 1] := 4.04460; fTable_Be[558, 2] := 0.0271914;
